			//Type Arrays
			//ARRAY OF BOOL
			IF FIND(Lynus_Standards.GVL_Communicator.arrInterfaceInfoAlVariables[byReadWriteArrayNumber,udiActiveNumberOfSymbol_ReadAds].sSymbolType,'OF BOOL') <> 0 THEN
				stADSRead_ReadAds[udiActiveNumberOfSymbol_ReadAds].sFullSymbolName := Lynus_Standards.GVL_Communicator.arrInterfaceInfoAlVariables[byReadWriteArrayNumber,udiActiveNumberOfSymbol_ReadAds].sFullSymbolName;
					stADSRead_ReadAds[udiActiveNumberOfSymbol_ReadAds].arrValue := arrValueDefault_ReadAds;	
						IF Lynus_Standards.GVL_Communicator.arrInterfaceInfoAlVariables[byReadWriteArrayNumber,udiActiveNumberOfSymbol_ReadAds].uiSizeArray <= Lynus_Standards.Constants_Communicator.bySizeOfValueArray THEN  
							FOR uiLPWriteValueByArray_ReadAds := 1 TO Lynus_Standards.GVL_Communicator.arrInterfaceInfoAlVariables[byReadWriteArrayNumber,udiActiveNumberOfSymbol_ReadAds].uiSizeArray BY 1 DO 	
								stADSRead_ReadAds[udiActiveNumberOfSymbol_ReadAds].arrValue[uiLPWriteValueByArray_ReadAds] := BYTE_TO_STRING(arrValueAfterRead_ReadAds[uiLPWriteValueByArray_ReadAds]);
							END_FOR 
						END_IF
			END_IF 
				//ARRAY OF BYTE
				IF FIND(Lynus_Standards.GVL_Communicator.arrInterfaceInfoAlVariables[byReadWriteArrayNumber,udiActiveNumberOfSymbol_ReadAds].sSymbolType,'OF BYTE') <> 0 THEN
					stADSRead_ReadAds[udiActiveNumberOfSymbol_ReadAds].sFullSymbolName := Lynus_Standards.GVL_Communicator.arrInterfaceInfoAlVariables[byReadWriteArrayNumber,udiActiveNumberOfSymbol_ReadAds].sFullSymbolName;
						stADSRead_ReadAds[udiActiveNumberOfSymbol_ReadAds].arrValue := arrValueDefault_ReadAds;	
							IF Lynus_Standards.GVL_Communicator.arrInterfaceInfoAlVariables[byReadWriteArrayNumber,udiActiveNumberOfSymbol_ReadAds].uiSizeArray <= Lynus_Standards.Constants_Communicator.bySizeOfValueArray THEN  
								FOR uiLPWriteValueByArray_ReadAds := 1 TO Lynus_Standards.GVL_Communicator.arrInterfaceInfoAlVariables[byReadWriteArrayNumber,udiActiveNumberOfSymbol_ReadAds].uiSizeArray BY 1 DO 	
									stADSRead_ReadAds[udiActiveNumberOfSymbol_ReadAds].arrValue[uiLPWriteValueByArray_ReadAds] := BYTE_TO_STRING(arrValueAfterRead_ReadAds[uiLPWriteValueByArray_ReadAds]);
								END_FOR 
							END_IF
				END_IF
			//ARRAY OF WORD
			IF FIND(Lynus_Standards.GVL_Communicator.arrInterfaceInfoAlVariables[byReadWriteArrayNumber,udiActiveNumberOfSymbol_ReadAds].sSymbolType,'OF WORD') <> 0 THEN
				stADSRead_ReadAds[udiActiveNumberOfSymbol_ReadAds].sFullSymbolName := Lynus_Standards.GVL_Communicator.arrInterfaceInfoAlVariables[byReadWriteArrayNumber,udiActiveNumberOfSymbol_ReadAds].sFullSymbolName;
					stADSRead_ReadAds[udiActiveNumberOfSymbol_ReadAds].arrValue := arrValueDefault_ReadAds;	
						IF Lynus_Standards.GVL_Communicator.arrInterfaceInfoAlVariables[byReadWriteArrayNumber,udiActiveNumberOfSymbol_ReadAds].uiSizeArray <= Lynus_Standards.Constants_Communicator.bySizeOfValueArray THEN  
							FOR uiLPWriteValueByArray_ReadAds := 1 TO Lynus_Standards.GVL_Communicator.arrInterfaceInfoAlVariables[byReadWriteArrayNumber,udiActiveNumberOfSymbol_ReadAds].uiSizeArray BY 1 DO
								arrCounterWriteValueInArray_ReadAds[1] := LIMIT(1,arrCounterWriteValueInArray_ReadAds[1],1600); arrCounterWriteValueInArray_ReadAds[2] := LIMIT(2,arrCounterWriteValueInArray_ReadAds[2],1600);
									stADSRead_ReadAds[udiActiveNumberOfSymbol_ReadAds].arrValue[uiLPWriteValueByArray_ReadAds] := WORD_TO_STRING(SHL(BYTE_TO_WORD(arrValueAfterRead_ReadAds[arrCounterWriteValueInArray_ReadAds[2]]),8) + BYTE_TO_WORD(arrValueAfterRead_ReadAds[arrCounterWriteValueInArray_ReadAds[1]]));;
								arrCounterWriteValueInArray_ReadAds[1] := arrCounterWriteValueInArray_ReadAds[1] + 2; arrCounterWriteValueInArray_ReadAds[2] := arrCounterWriteValueInArray_ReadAds[2] + 2;
							END_FOR 
						END_IF
			END_IF
				//ARRAY OF DWORD	
				IF FIND(Lynus_Standards.GVL_Communicator.arrInterfaceInfoAlVariables[byReadWriteArrayNumber,udiActiveNumberOfSymbol_ReadAds].sSymbolType,'OF DWORD') <> 0 THEN
					stADSRead_ReadAds[udiActiveNumberOfSymbol_ReadAds].sFullSymbolName := Lynus_Standards.GVL_Communicator.arrInterfaceInfoAlVariables[byReadWriteArrayNumber,udiActiveNumberOfSymbol_ReadAds].sFullSymbolName;
						stADSRead_ReadAds[udiActiveNumberOfSymbol_ReadAds].arrValue := arrValueDefault_ReadAds;	
							IF Lynus_Standards.GVL_Communicator.arrInterfaceInfoAlVariables[byReadWriteArrayNumber,udiActiveNumberOfSymbol_ReadAds].uiSizeArray <= Lynus_Standards.Constants_Communicator.bySizeOfValueArray THEN  
								FOR uiLPWriteValueByArray_ReadAds := 1 TO Lynus_Standards.GVL_Communicator.arrInterfaceInfoAlVariables[byReadWriteArrayNumber,udiActiveNumberOfSymbol_ReadAds].uiSizeArray BY 1 DO
									arrCounterWriteValueInArray_ReadAds[1] := LIMIT(1,arrCounterWriteValueInArray_ReadAds[1],1600); arrCounterWriteValueInArray_ReadAds[2] := LIMIT(2,arrCounterWriteValueInArray_ReadAds[2],1600);
										arrCounterWriteValueInArray_ReadAds[3] := LIMIT(3,arrCounterWriteValueInArray_ReadAds[3],1600); arrCounterWriteValueInArray_ReadAds[4] := LIMIT(4,arrCounterWriteValueInArray_ReadAds[4],1600);
											stADSRead_ReadAds[udiActiveNumberOfSymbol_ReadAds].arrValue[uiLPWriteValueByArray_ReadAds] := DWORD_TO_STRING(SHL(BYTE_TO_DWORD(arrValueAfterRead_ReadAds[arrCounterWriteValueInArray_ReadAds[4]]),24) + SHL(BYTE_TO_DWORD(arrValueAfterRead_ReadAds[arrCounterWriteValueInArray_ReadAds[3]]),16) + SHL(BYTE_TO_DWORD(arrValueAfterRead_ReadAds[arrCounterWriteValueInArray_ReadAds[2]]),8) + BYTE_TO_DWORD(arrValueAfterRead_ReadAds[arrCounterWriteValueInArray_ReadAds[1]]));
									arrCounterWriteValueInArray_ReadAds[1] := arrCounterWriteValueInArray_ReadAds[1] + 4; arrCounterWriteValueInArray_ReadAds[2] := arrCounterWriteValueInArray_ReadAds[2] + 4;
										arrCounterWriteValueInArray_ReadAds[3] := arrCounterWriteValueInArray_ReadAds[3] + 4; arrCounterWriteValueInArray_ReadAds[4] := arrCounterWriteValueInArray_ReadAds[4] + 4;
								END_FOR 
							END_IF
				END_IF
			//ARRAY OF SINT
			IF FIND(Lynus_Standards.GVL_Communicator.arrInterfaceInfoAlVariables[byReadWriteArrayNumber,udiActiveNumberOfSymbol_ReadAds].sSymbolType,'OF SINT') <> 0 THEN
				stADSRead_ReadAds[udiActiveNumberOfSymbol_ReadAds].sFullSymbolName := Lynus_Standards.GVL_Communicator.arrInterfaceInfoAlVariables[byReadWriteArrayNumber,udiActiveNumberOfSymbol_ReadAds].sFullSymbolName;
					stADSRead_ReadAds[udiActiveNumberOfSymbol_ReadAds].arrValue := arrValueDefault_ReadAds;	
						IF Lynus_Standards.GVL_Communicator.arrInterfaceInfoAlVariables[byReadWriteArrayNumber,udiActiveNumberOfSymbol_ReadAds].uiSizeArray <= Lynus_Standards.Constants_Communicator.bySizeOfValueArray THEN  
							FOR uiLPWriteValueByArray_ReadAds := 1 TO Lynus_Standards.GVL_Communicator.arrInterfaceInfoAlVariables[byReadWriteArrayNumber,udiActiveNumberOfSymbol_ReadAds].uiSizeArray BY 1 DO 	
								stADSRead_ReadAds[udiActiveNumberOfSymbol_ReadAds].arrValue[uiLPWriteValueByArray_ReadAds] := SINT_TO_STRING(BYTE_TO_SINT(arrValueAfterRead_ReadAds[uiLPWriteValueByArray_ReadAds]));
							END_FOR 
						END_IF
			END_IF
				//ARRAY OF USINT
				IF FIND(Lynus_Standards.GVL_Communicator.arrInterfaceInfoAlVariables[byReadWriteArrayNumber,udiActiveNumberOfSymbol_ReadAds].sSymbolType,'OF USINT') <> 0 THEN
					stADSRead_ReadAds[udiActiveNumberOfSymbol_ReadAds].sFullSymbolName := Lynus_Standards.GVL_Communicator.arrInterfaceInfoAlVariables[byReadWriteArrayNumber,udiActiveNumberOfSymbol_ReadAds].sFullSymbolName;
						stADSRead_ReadAds[udiActiveNumberOfSymbol_ReadAds].arrValue := arrValueDefault_ReadAds;	
							IF Lynus_Standards.GVL_Communicator.arrInterfaceInfoAlVariables[byReadWriteArrayNumber,udiActiveNumberOfSymbol_ReadAds].uiSizeArray <= Lynus_Standards.Constants_Communicator.bySizeOfValueArray THEN  
								FOR uiLPWriteValueByArray_ReadAds := 1 TO Lynus_Standards.GVL_Communicator.arrInterfaceInfoAlVariables[byReadWriteArrayNumber,udiActiveNumberOfSymbol_ReadAds].uiSizeArray BY 1 DO 	
									stADSRead_ReadAds[udiActiveNumberOfSymbol_ReadAds].arrValue[uiLPWriteValueByArray_ReadAds] := USINT_TO_STRING(BYTE_TO_USINT(arrValueAfterRead_ReadAds[uiLPWriteValueByArray_ReadAds]));
								END_FOR 
							END_IF
				END_IF
			//ARRAY OF INT
			IF FIND(Lynus_Standards.GVL_Communicator.arrInterfaceInfoAlVariables[byReadWriteArrayNumber,udiActiveNumberOfSymbol_ReadAds].sSymbolType,'OF INT') <> 0 THEN
				stADSRead_ReadAds[udiActiveNumberOfSymbol_ReadAds].sFullSymbolName := Lynus_Standards.GVL_Communicator.arrInterfaceInfoAlVariables[byReadWriteArrayNumber,udiActiveNumberOfSymbol_ReadAds].sFullSymbolName;
					stADSRead_ReadAds[udiActiveNumberOfSymbol_ReadAds].arrValue := arrValueDefault_ReadAds;	
						IF Lynus_Standards.GVL_Communicator.arrInterfaceInfoAlVariables[byReadWriteArrayNumber,udiActiveNumberOfSymbol_ReadAds].uiSizeArray <= Lynus_Standards.Constants_Communicator.bySizeOfValueArray THEN  
							FOR uiLPWriteValueByArray_ReadAds := 1 TO Lynus_Standards.GVL_Communicator.arrInterfaceInfoAlVariables[byReadWriteArrayNumber,udiActiveNumberOfSymbol_ReadAds].uiSizeArray BY 1 DO
								arrCounterWriteValueInArray_ReadAds[1] := LIMIT(1,arrCounterWriteValueInArray_ReadAds[1],1600); arrCounterWriteValueInArray_ReadAds[2] := LIMIT(2,arrCounterWriteValueInArray_ReadAds[2],1600);
									stADSRead_ReadAds[udiActiveNumberOfSymbol_ReadAds].arrValue[uiLPWriteValueByArray_ReadAds] := INT_TO_STRING(SHL(BYTE_TO_INT(arrValueAfterRead_ReadAds[arrCounterWriteValueInArray_ReadAds[2]]),8) + BYTE_TO_INT(arrValueAfterRead_ReadAds[arrCounterWriteValueInArray_ReadAds[1]]));;
								arrCounterWriteValueInArray_ReadAds[1] := arrCounterWriteValueInArray_ReadAds[1] + 2; arrCounterWriteValueInArray_ReadAds[2] := arrCounterWriteValueInArray_ReadAds[2] + 2;
							END_FOR 
						END_IF
			END_IF
				//ARRAY OF UINT
				IF FIND(Lynus_Standards.GVL_Communicator.arrInterfaceInfoAlVariables[byReadWriteArrayNumber,udiActiveNumberOfSymbol_ReadAds].sSymbolType,'OF UINT') <> 0 THEN
					stADSRead_ReadAds[udiActiveNumberOfSymbol_ReadAds].sFullSymbolName := Lynus_Standards.GVL_Communicator.arrInterfaceInfoAlVariables[byReadWriteArrayNumber,udiActiveNumberOfSymbol_ReadAds].sFullSymbolName;
						stADSRead_ReadAds[udiActiveNumberOfSymbol_ReadAds].arrValue := arrValueDefault_ReadAds;	
							IF Lynus_Standards.GVL_Communicator.arrInterfaceInfoAlVariables[byReadWriteArrayNumber,udiActiveNumberOfSymbol_ReadAds].uiSizeArray <= Lynus_Standards.Constants_Communicator.bySizeOfValueArray THEN  
								FOR uiLPWriteValueByArray_ReadAds := 1 TO Lynus_Standards.GVL_Communicator.arrInterfaceInfoAlVariables[byReadWriteArrayNumber,udiActiveNumberOfSymbol_ReadAds].uiSizeArray BY 1 DO
									arrCounterWriteValueInArray_ReadAds[1] := LIMIT(1,arrCounterWriteValueInArray_ReadAds[1],1600); arrCounterWriteValueInArray_ReadAds[2] := LIMIT(2,arrCounterWriteValueInArray_ReadAds[2],1600);
										stADSRead_ReadAds[udiActiveNumberOfSymbol_ReadAds].arrValue[uiLPWriteValueByArray_ReadAds] := UINT_TO_STRING(SHL(BYTE_TO_UINT(arrValueAfterRead_ReadAds[arrCounterWriteValueInArray_ReadAds[2]]),8) + BYTE_TO_UINT(arrValueAfterRead_ReadAds[arrCounterWriteValueInArray_ReadAds[1]]));;
									arrCounterWriteValueInArray_ReadAds[1] := arrCounterWriteValueInArray_ReadAds[1] + 2; arrCounterWriteValueInArray_ReadAds[2] := arrCounterWriteValueInArray_ReadAds[2] + 2;
								END_FOR 
							END_IF
				END_IF
			//ARRAY OF DINT	
			IF FIND(Lynus_Standards.GVL_Communicator.arrInterfaceInfoAlVariables[byReadWriteArrayNumber,udiActiveNumberOfSymbol_ReadAds].sSymbolType,'OF DINT') <> 0 THEN
				stADSRead_ReadAds[udiActiveNumberOfSymbol_ReadAds].sFullSymbolName := Lynus_Standards.GVL_Communicator.arrInterfaceInfoAlVariables[byReadWriteArrayNumber,udiActiveNumberOfSymbol_ReadAds].sFullSymbolName;
					stADSRead_ReadAds[udiActiveNumberOfSymbol_ReadAds].arrValue := arrValueDefault_ReadAds;	
						IF Lynus_Standards.GVL_Communicator.arrInterfaceInfoAlVariables[byReadWriteArrayNumber,udiActiveNumberOfSymbol_ReadAds].uiSizeArray <= Lynus_Standards.Constants_Communicator.bySizeOfValueArray THEN  
							FOR uiLPWriteValueByArray_ReadAds := 1 TO Lynus_Standards.GVL_Communicator.arrInterfaceInfoAlVariables[byReadWriteArrayNumber,udiActiveNumberOfSymbol_ReadAds].uiSizeArray BY 1 DO
								arrCounterWriteValueInArray_ReadAds[1] := LIMIT(1,arrCounterWriteValueInArray_ReadAds[1],1600); arrCounterWriteValueInArray_ReadAds[2] := LIMIT(2,arrCounterWriteValueInArray_ReadAds[2],1600);
									arrCounterWriteValueInArray_ReadAds[3] := LIMIT(3,arrCounterWriteValueInArray_ReadAds[3],1600); arrCounterWriteValueInArray_ReadAds[4] := LIMIT(4,arrCounterWriteValueInArray_ReadAds[4],1600);
										stADSRead_ReadAds[udiActiveNumberOfSymbol_ReadAds].arrValue[uiLPWriteValueByArray_ReadAds] := DINT_TO_STRING(SHL(BYTE_TO_DINT(arrValueAfterRead_ReadAds[arrCounterWriteValueInArray_ReadAds[4]]),24) + SHL(BYTE_TO_DINT(arrValueAfterRead_ReadAds[arrCounterWriteValueInArray_ReadAds[3]]),16) + SHL(BYTE_TO_DINT(arrValueAfterRead_ReadAds[arrCounterWriteValueInArray_ReadAds[2]]),8) + BYTE_TO_DINT(arrValueAfterRead_ReadAds[arrCounterWriteValueInArray_ReadAds[1]]));
								arrCounterWriteValueInArray_ReadAds[1] := arrCounterWriteValueInArray_ReadAds[1] + 4; arrCounterWriteValueInArray_ReadAds[2] := arrCounterWriteValueInArray_ReadAds[2] + 4;
									arrCounterWriteValueInArray_ReadAds[3] := arrCounterWriteValueInArray_ReadAds[3] + 4; arrCounterWriteValueInArray_ReadAds[4] := arrCounterWriteValueInArray_ReadAds[4] + 4;
							END_FOR 
						END_IF
			END_IF
				//ARRAY OF UDINT	
				IF FIND(Lynus_Standards.GVL_Communicator.arrInterfaceInfoAlVariables[byReadWriteArrayNumber,udiActiveNumberOfSymbol_ReadAds].sSymbolType,'OF UDINT') <> 0 THEN
					stADSRead_ReadAds[udiActiveNumberOfSymbol_ReadAds].sFullSymbolName := Lynus_Standards.GVL_Communicator.arrInterfaceInfoAlVariables[byReadWriteArrayNumber,udiActiveNumberOfSymbol_ReadAds].sFullSymbolName;
						stADSRead_ReadAds[udiActiveNumberOfSymbol_ReadAds].arrValue := arrValueDefault_ReadAds;	
							IF Lynus_Standards.GVL_Communicator.arrInterfaceInfoAlVariables[byReadWriteArrayNumber,udiActiveNumberOfSymbol_ReadAds].uiSizeArray <= Lynus_Standards.Constants_Communicator.bySizeOfValueArray THEN  
								FOR uiLPWriteValueByArray_ReadAds := 1 TO Lynus_Standards.GVL_Communicator.arrInterfaceInfoAlVariables[byReadWriteArrayNumber,udiActiveNumberOfSymbol_ReadAds].uiSizeArray BY 1 DO
									arrCounterWriteValueInArray_ReadAds[1] := LIMIT(1,arrCounterWriteValueInArray_ReadAds[1],1600); arrCounterWriteValueInArray_ReadAds[2] := LIMIT(2,arrCounterWriteValueInArray_ReadAds[2],1600);
										arrCounterWriteValueInArray_ReadAds[3] := LIMIT(3,arrCounterWriteValueInArray_ReadAds[3],1600); arrCounterWriteValueInArray_ReadAds[4] := LIMIT(4,arrCounterWriteValueInArray_ReadAds[4],1600);
											stADSRead_ReadAds[udiActiveNumberOfSymbol_ReadAds].arrValue[uiLPWriteValueByArray_ReadAds] := UDINT_TO_STRING(SHL(BYTE_TO_UDINT(arrValueAfterRead_ReadAds[arrCounterWriteValueInArray_ReadAds[4]]),24) + SHL(BYTE_TO_UDINT(arrValueAfterRead_ReadAds[arrCounterWriteValueInArray_ReadAds[3]]),16) + SHL(BYTE_TO_UDINT(arrValueAfterRead_ReadAds[arrCounterWriteValueInArray_ReadAds[2]]),8) + BYTE_TO_UDINT(arrValueAfterRead_ReadAds[arrCounterWriteValueInArray_ReadAds[1]]));
									arrCounterWriteValueInArray_ReadAds[1] := arrCounterWriteValueInArray_ReadAds[1] + 4; arrCounterWriteValueInArray_ReadAds[2] := arrCounterWriteValueInArray_ReadAds[2] + 4;
										arrCounterWriteValueInArray_ReadAds[3] := arrCounterWriteValueInArray_ReadAds[3] + 4; arrCounterWriteValueInArray_ReadAds[4] := arrCounterWriteValueInArray_ReadAds[4] + 4;
								END_FOR 
							END_IF
				END_IF
					//ARRAY OF LINT	
					IF FIND(Lynus_Standards.GVL_Communicator.arrInterfaceInfoAlVariables[byReadWriteArrayNumber,udiActiveNumberOfSymbol_ReadAds].sSymbolType,'OF LINT') <> 0 THEN
						stADSRead_ReadAds[udiActiveNumberOfSymbol_ReadAds].sFullSymbolName := Lynus_Standards.GVL_Communicator.arrInterfaceInfoAlVariables[byReadWriteArrayNumber,udiActiveNumberOfSymbol_ReadAds].sFullSymbolName;
							stADSRead_ReadAds[udiActiveNumberOfSymbol_ReadAds].arrValue := arrValueDefault_ReadAds;	
								IF Lynus_Standards.GVL_Communicator.arrInterfaceInfoAlVariables[byReadWriteArrayNumber,udiActiveNumberOfSymbol_ReadAds].uiSizeArray <= Lynus_Standards.Constants_Communicator.bySizeOfValueArray THEN  
									FOR uiLPWriteValueByArray_ReadAds := 1 TO Lynus_Standards.GVL_Communicator.arrInterfaceInfoAlVariables[byReadWriteArrayNumber,udiActiveNumberOfSymbol_ReadAds].uiSizeArray BY 1 DO
										arrCounterWriteValueInArray_ReadAds[1] := LIMIT(1,arrCounterWriteValueInArray_ReadAds[1],1600); arrCounterWriteValueInArray_ReadAds[2] := LIMIT(2,arrCounterWriteValueInArray_ReadAds[2],1600);
											arrCounterWriteValueInArray_ReadAds[3] := LIMIT(3,arrCounterWriteValueInArray_ReadAds[3],1600); arrCounterWriteValueInArray_ReadAds[4] := LIMIT(4,arrCounterWriteValueInArray_ReadAds[4],1600);
												arrCounterWriteValueInArray_ReadAds[5] := LIMIT(5,arrCounterWriteValueInArray_ReadAds[5],1600); arrCounterWriteValueInArray_ReadAds[6] := LIMIT(6,arrCounterWriteValueInArray_ReadAds[6],1600);
													arrCounterWriteValueInArray_ReadAds[7] := LIMIT(7,arrCounterWriteValueInArray_ReadAds[7],1600); arrCounterWriteValueInArray_ReadAds[8] := LIMIT(8,arrCounterWriteValueInArray_ReadAds[8],1600);
														stADSRead_ReadAds[udiActiveNumberOfSymbol_ReadAds].arrValue[uiLPWriteValueByArray_ReadAds] := LINT_TO_STRING(SHL(BYTE_TO_LINT(arrValueAfterRead_ReadAds[arrCounterWriteValueInArray_ReadAds[8]]),56) + SHL(BYTE_TO_LINT(arrValueAfterRead_ReadAds[arrCounterWriteValueInArray_ReadAds[7]]),48) + SHL(BYTE_TO_LINT(arrValueAfterRead_ReadAds[arrCounterWriteValueInArray_ReadAds[6]]),40) + SHL(BYTE_TO_LINT(arrValueAfterRead_ReadAds[arrCounterWriteValueInArray_ReadAds[5]]),32) +
																																							SHL(BYTE_TO_LINT(arrValueAfterRead_ReadAds[arrCounterWriteValueInArray_ReadAds[4]]),24) + SHL(BYTE_TO_LINT(arrValueAfterRead_ReadAds[arrCounterWriteValueInArray_ReadAds[3]]),16) + SHL(BYTE_TO_LINT(arrValueAfterRead_ReadAds[arrCounterWriteValueInArray_ReadAds[2]]),8) + BYTE_TO_LINT(arrValueAfterRead_ReadAds[arrCounterWriteValueInArray_ReadAds[1]]));
										arrCounterWriteValueInArray_ReadAds[1] := arrCounterWriteValueInArray_ReadAds[1] + 8; arrCounterWriteValueInArray_ReadAds[2] := arrCounterWriteValueInArray_ReadAds[2] + 8;
											arrCounterWriteValueInArray_ReadAds[3] := arrCounterWriteValueInArray_ReadAds[3] + 8; arrCounterWriteValueInArray_ReadAds[4] := arrCounterWriteValueInArray_ReadAds[4] + 8;
												arrCounterWriteValueInArray_ReadAds[5] := arrCounterWriteValueInArray_ReadAds[5] + 8; arrCounterWriteValueInArray_ReadAds[6] := arrCounterWriteValueInArray_ReadAds[6] + 8;
													arrCounterWriteValueInArray_ReadAds[7] := arrCounterWriteValueInArray_ReadAds[7] + 8; arrCounterWriteValueInArray_ReadAds[8] := arrCounterWriteValueInArray_ReadAds[8] + 8;
									END_FOR 
								END_IF
					END_IF
				//ARRAY OF ULINT	
				IF FIND(Lynus_Standards.GVL_Communicator.arrInterfaceInfoAlVariables[byReadWriteArrayNumber,udiActiveNumberOfSymbol_ReadAds].sSymbolType,'OF ULINT') <> 0 THEN
					stADSRead_ReadAds[udiActiveNumberOfSymbol_ReadAds].sFullSymbolName := Lynus_Standards.GVL_Communicator.arrInterfaceInfoAlVariables[byReadWriteArrayNumber,udiActiveNumberOfSymbol_ReadAds].sFullSymbolName;
						stADSRead_ReadAds[udiActiveNumberOfSymbol_ReadAds].arrValue := arrValueDefault_ReadAds;	
							IF Lynus_Standards.GVL_Communicator.arrInterfaceInfoAlVariables[byReadWriteArrayNumber,udiActiveNumberOfSymbol_ReadAds].uiSizeArray <= Lynus_Standards.Constants_Communicator.bySizeOfValueArray THEN  
								FOR uiLPWriteValueByArray_ReadAds := 1 TO Lynus_Standards.GVL_Communicator.arrInterfaceInfoAlVariables[byReadWriteArrayNumber,udiActiveNumberOfSymbol_ReadAds].uiSizeArray BY 1 DO
									arrCounterWriteValueInArray_ReadAds[1] := LIMIT(1,arrCounterWriteValueInArray_ReadAds[1],1600); arrCounterWriteValueInArray_ReadAds[2] := LIMIT(2,arrCounterWriteValueInArray_ReadAds[2],1600);
										arrCounterWriteValueInArray_ReadAds[3] := LIMIT(3,arrCounterWriteValueInArray_ReadAds[3],1600); arrCounterWriteValueInArray_ReadAds[4] := LIMIT(4,arrCounterWriteValueInArray_ReadAds[4],1600);
											arrCounterWriteValueInArray_ReadAds[5] := LIMIT(5,arrCounterWriteValueInArray_ReadAds[5],1600); arrCounterWriteValueInArray_ReadAds[6] := LIMIT(6,arrCounterWriteValueInArray_ReadAds[6],1600);
												arrCounterWriteValueInArray_ReadAds[7] := LIMIT(7,arrCounterWriteValueInArray_ReadAds[7],1600); arrCounterWriteValueInArray_ReadAds[8] := LIMIT(8,arrCounterWriteValueInArray_ReadAds[8],1600);
													stADSRead_ReadAds[udiActiveNumberOfSymbol_ReadAds].arrValue[uiLPWriteValueByArray_ReadAds] := ULINT_TO_STRING(SHL(BYTE_TO_ULINT(arrValueAfterRead_ReadAds[arrCounterWriteValueInArray_ReadAds[8]]),56) + SHL(BYTE_TO_ULINT(arrValueAfterRead_ReadAds[arrCounterWriteValueInArray_ReadAds[7]]),48) + SHL(BYTE_TO_ULINT(arrValueAfterRead_ReadAds[arrCounterWriteValueInArray_ReadAds[6]]),40) + SHL(BYTE_TO_ULINT(arrValueAfterRead_ReadAds[arrCounterWriteValueInArray_ReadAds[5]]),32) +
																																						SHL(BYTE_TO_ULINT(arrValueAfterRead_ReadAds[arrCounterWriteValueInArray_ReadAds[4]]),24) + SHL(BYTE_TO_ULINT(arrValueAfterRead_ReadAds[arrCounterWriteValueInArray_ReadAds[3]]),16) + SHL(BYTE_TO_ULINT(arrValueAfterRead_ReadAds[arrCounterWriteValueInArray_ReadAds[2]]),8) + BYTE_TO_ULINT(arrValueAfterRead_ReadAds[arrCounterWriteValueInArray_ReadAds[1]]));
									arrCounterWriteValueInArray_ReadAds[1] := arrCounterWriteValueInArray_ReadAds[1] + 8; arrCounterWriteValueInArray_ReadAds[2] := arrCounterWriteValueInArray_ReadAds[2] + 8;
										arrCounterWriteValueInArray_ReadAds[3] := arrCounterWriteValueInArray_ReadAds[3] + 8; arrCounterWriteValueInArray_ReadAds[4] := arrCounterWriteValueInArray_ReadAds[4] + 8;
											arrCounterWriteValueInArray_ReadAds[5] := arrCounterWriteValueInArray_ReadAds[5] + 8; arrCounterWriteValueInArray_ReadAds[6] := arrCounterWriteValueInArray_ReadAds[6] + 8;
												arrCounterWriteValueInArray_ReadAds[7] := arrCounterWriteValueInArray_ReadAds[7] + 8; arrCounterWriteValueInArray_ReadAds[8] := arrCounterWriteValueInArray_ReadAds[8] + 8;
								END_FOR 
							END_IF
				END_IF
					//ARRAY OF LWORD	
					IF FIND(Lynus_Standards.GVL_Communicator.arrInterfaceInfoAlVariables[byReadWriteArrayNumber,udiActiveNumberOfSymbol_ReadAds].sSymbolType,'OF LWORD') <> 0 THEN
						stADSRead_ReadAds[udiActiveNumberOfSymbol_ReadAds].sFullSymbolName := Lynus_Standards.GVL_Communicator.arrInterfaceInfoAlVariables[byReadWriteArrayNumber,udiActiveNumberOfSymbol_ReadAds].sFullSymbolName;
							stADSRead_ReadAds[udiActiveNumberOfSymbol_ReadAds].arrValue := arrValueDefault_ReadAds;	
								IF Lynus_Standards.GVL_Communicator.arrInterfaceInfoAlVariables[byReadWriteArrayNumber,udiActiveNumberOfSymbol_ReadAds].uiSizeArray <= Lynus_Standards.Constants_Communicator.bySizeOfValueArray THEN  
									FOR uiLPWriteValueByArray_ReadAds := 1 TO Lynus_Standards.GVL_Communicator.arrInterfaceInfoAlVariables[byReadWriteArrayNumber,udiActiveNumberOfSymbol_ReadAds].uiSizeArray BY 1 DO
										arrCounterWriteValueInArray_ReadAds[1] := LIMIT(1,arrCounterWriteValueInArray_ReadAds[1],1600); arrCounterWriteValueInArray_ReadAds[2] := LIMIT(2,arrCounterWriteValueInArray_ReadAds[2],1600);
											arrCounterWriteValueInArray_ReadAds[3] := LIMIT(3,arrCounterWriteValueInArray_ReadAds[3],1600); arrCounterWriteValueInArray_ReadAds[4] := LIMIT(4,arrCounterWriteValueInArray_ReadAds[4],1600);
												arrCounterWriteValueInArray_ReadAds[5] := LIMIT(5,arrCounterWriteValueInArray_ReadAds[5],1600); arrCounterWriteValueInArray_ReadAds[6] := LIMIT(6,arrCounterWriteValueInArray_ReadAds[6],1600);
													arrCounterWriteValueInArray_ReadAds[7] := LIMIT(7,arrCounterWriteValueInArray_ReadAds[7],1600); arrCounterWriteValueInArray_ReadAds[8] := LIMIT(8,arrCounterWriteValueInArray_ReadAds[8],1600);
														stADSRead_ReadAds[udiActiveNumberOfSymbol_ReadAds].arrValue[uiLPWriteValueByArray_ReadAds] := LWORD_TO_STRING(SHL(BYTE_TO_LWORD(arrValueAfterRead_ReadAds[arrCounterWriteValueInArray_ReadAds[8]]),56) + SHL(BYTE_TO_LWORD(arrValueAfterRead_ReadAds[arrCounterWriteValueInArray_ReadAds[7]]),48) + SHL(BYTE_TO_LWORD(arrValueAfterRead_ReadAds[arrCounterWriteValueInArray_ReadAds[6]]),40) + SHL(BYTE_TO_LWORD(arrValueAfterRead_ReadAds[arrCounterWriteValueInArray_ReadAds[5]]),32) +
																																							SHL(BYTE_TO_LWORD(arrValueAfterRead_ReadAds[arrCounterWriteValueInArray_ReadAds[4]]),24) + SHL(BYTE_TO_LWORD(arrValueAfterRead_ReadAds[arrCounterWriteValueInArray_ReadAds[3]]),16) + SHL(BYTE_TO_LWORD(arrValueAfterRead_ReadAds[arrCounterWriteValueInArray_ReadAds[2]]),8) + BYTE_TO_LWORD(arrValueAfterRead_ReadAds[arrCounterWriteValueInArray_ReadAds[1]]));
										arrCounterWriteValueInArray_ReadAds[1] := arrCounterWriteValueInArray_ReadAds[1] + 8; arrCounterWriteValueInArray_ReadAds[2] := arrCounterWriteValueInArray_ReadAds[2] + 8;
											arrCounterWriteValueInArray_ReadAds[3] := arrCounterWriteValueInArray_ReadAds[3] + 8; arrCounterWriteValueInArray_ReadAds[4] := arrCounterWriteValueInArray_ReadAds[4] + 8;
												arrCounterWriteValueInArray_ReadAds[5] := arrCounterWriteValueInArray_ReadAds[5] + 8; arrCounterWriteValueInArray_ReadAds[6] := arrCounterWriteValueInArray_ReadAds[6] + 8;
													arrCounterWriteValueInArray_ReadAds[7] := arrCounterWriteValueInArray_ReadAds[7] + 8; arrCounterWriteValueInArray_ReadAds[8] := arrCounterWriteValueInArray_ReadAds[8] + 8;
									END_FOR 
								END_IF
					END_IF
				//ARRAY OF REAL
				IF FIND(Lynus_Standards.GVL_Communicator.arrInterfaceInfoAlVariables[byReadWriteArrayNumber,udiActiveNumberOfSymbol_ReadAds].sSymbolType,'OF REAL') <> 0 THEN
					stADSRead_ReadAds[udiActiveNumberOfSymbol_ReadAds].sFullSymbolName := Lynus_Standards.GVL_Communicator.arrInterfaceInfoAlVariables[byReadWriteArrayNumber,udiActiveNumberOfSymbol_ReadAds].sFullSymbolName;
						stADSRead_ReadAds[udiActiveNumberOfSymbol_ReadAds].arrValue := arrValueDefault_ReadAds;	
							IF Lynus_Standards.GVL_Communicator.arrInterfaceInfoAlVariables[byReadWriteArrayNumber,udiActiveNumberOfSymbol_ReadAds].uiSizeArray <= Lynus_Standards.Constants_Communicator.bySizeOfValueArray THEN  
								FOR uiLPWriteValueByArray_ReadAds := 1 TO Lynus_Standards.GVL_Communicator.arrInterfaceInfoAlVariables[byReadWriteArrayNumber,udiActiveNumberOfSymbol_ReadAds].uiSizeArray BY 1 DO
									arrCounterWriteValueInArray_ReadAds[1] := LIMIT(1,arrCounterWriteValueInArray_ReadAds[1],1600); arrCounterWriteValueInArray_ReadAds[2] := LIMIT(2,arrCounterWriteValueInArray_ReadAds[2],1600);
										arrCounterWriteValueInArray_ReadAds[3] := LIMIT(3,arrCounterWriteValueInArray_ReadAds[3],1600); arrCounterWriteValueInArray_ReadAds[4] := LIMIT(4,arrCounterWriteValueInArray_ReadAds[4],1600);
											unConvertDWORD_TO_REAL_ReadAds.dwRawValue := DINT_TO_DWORD(DWORD_TO_DINT(SHL(BYTE_TO_DWORD(arrValueAfterRead_ReadAds[arrCounterWriteValueInArray_ReadAds[4]]),24) + SHL(BYTE_TO_DWORD(arrValueAfterRead_ReadAds[arrCounterWriteValueInArray_ReadAds[3]]),16) + SHL(BYTE_TO_DWORD(arrValueAfterRead_ReadAds[arrCounterWriteValueInArray_ReadAds[2]]),8) + BYTE_TO_DWORD(arrValueAfterRead_ReadAds[arrCounterWriteValueInArray_ReadAds[1]])));
									arrCounterWriteValueInArray_ReadAds[1] := arrCounterWriteValueInArray_ReadAds[1] + 4; arrCounterWriteValueInArray_ReadAds[2] := arrCounterWriteValueInArray_ReadAds[2] + 4;
										arrCounterWriteValueInArray_ReadAds[3] := arrCounterWriteValueInArray_ReadAds[3] + 4; arrCounterWriteValueInArray_ReadAds[4] := arrCounterWriteValueInArray_ReadAds[4] + 4;					
											IF IsFinite(F_REAL(unConvertDWORD_TO_REAL_ReadAds.rValueFloat)) THEN 
												IF LEN(REAL_TO_STRING(unConvertDWORD_TO_REAL_ReadAds.rValueFloat)) <= 30 THEN 
													IF FIND(REAL_TO_STRING(unConvertDWORD_TO_REAL_ReadAds.rValueFloat),'e') = 0 AND FIND(REAL_TO_STRING(unConvertDWORD_TO_REAL_ReadAds.rValueFloat),'E') = 0 THEN 
														sStringFloat_ReadAds := REAL_TO_STRING(unConvertDWORD_TO_REAL_ReadAds.rValueFloat);
															iFindPointFloat_ReadAds := FIND(sStringFloat_ReadAds,'.');
																sStringFloat_ReadAds := DELETE(sStringFloat_ReadAds,iFindPointFloat_ReadAds,1);
																	iPrecision_ReadAds := LEN(sStringFloat_ReadAds);
																		iPrecision_ReadAds := LIMIT(0,iPrecision_ReadAds,8);
														IF LEN(LREAL_TO_FMTSTR(REAL_TO_LREAL(unConvertDWORD_TO_REAL_ReadAds.rValueFloat),iPrecision_ReadAds,TRUE)) <= 30 THEN	 			
															//Check if the output from Function LREAL_TO_FMTSTR is ok 
															IF LREAL_TO_FMTSTR(REAL_TO_LREAL(unConvertDWORD_TO_REAL_ReadAds.rValueFloat),iPrecision_ReadAds,TRUE) <> '#INF' AND LREAL_TO_FMTSTR(REAL_TO_LREAL(unConvertDWORD_TO_REAL_ReadAds.rValueFloat),iPrecision_ReadAds,TRUE) <> '-#INF' AND
																LREAL_TO_FMTSTR(REAL_TO_LREAL(unConvertDWORD_TO_REAL_ReadAds.rValueFloat),iPrecision_ReadAds,TRUE) <> '#QNAN' AND LREAL_TO_FMTSTR(REAL_TO_LREAL(unConvertDWORD_TO_REAL_ReadAds.rValueFloat),iPrecision_ReadAds,TRUE) <> '-#QNAN' AND
																	LREAL_TO_FMTSTR(REAL_TO_LREAL(unConvertDWORD_TO_REAL_ReadAds.rValueFloat),iPrecision_ReadAds,TRUE) <> '#OVF' AND LREAL_TO_FMTSTR(REAL_TO_LREAL(unConvertDWORD_TO_REAL_ReadAds.rValueFloat),iPrecision_ReadAds,TRUE) <> '-#OVF' THEN	   	 			
																		stADSRead_ReadAds[udiActiveNumberOfSymbol_ReadAds].arrValue[uiLPWriteValueByArray_ReadAds] := LREAL_TO_FMTSTR(REAL_TO_LREAL(unConvertDWORD_TO_REAL_ReadAds.rValueFloat),iPrecision_ReadAds,TRUE);
															ELSE
																iState_ReadAds := 200;
																	uiInternError_ReadAds := 1;
															END_IF
														ELSE
															//Check if the output from Function LREAL_TO_FMTSTR is ok 
															IF MID(LREAL_TO_FMTSTR(REAL_TO_LREAL(unConvertDWORD_TO_REAL_ReadAds.rValueFloat),iPrecision_ReadAds,TRUE),30,1) <> '#INF' AND MID(LREAL_TO_FMTSTR(REAL_TO_LREAL(unConvertDWORD_TO_REAL_ReadAds.rValueFloat),iPrecision_ReadAds,TRUE),30,1) <> '-#INF' AND
																MID(LREAL_TO_FMTSTR(REAL_TO_LREAL(unConvertDWORD_TO_REAL_ReadAds.rValueFloat),iPrecision_ReadAds,TRUE),30,1) <> '#QNAN' AND MID(LREAL_TO_FMTSTR(REAL_TO_LREAL(unConvertDWORD_TO_REAL_ReadAds.rValueFloat),iPrecision_ReadAds,TRUE),30,1) <> '-#QNAN' AND
																	MID(LREAL_TO_FMTSTR(REAL_TO_LREAL(unConvertDWORD_TO_REAL_ReadAds.rValueFloat),iPrecision_ReadAds,TRUE),30,1) <> '#OVF' AND MID(LREAL_TO_FMTSTR(REAL_TO_LREAL(unConvertDWORD_TO_REAL_ReadAds.rValueFloat),iPrecision_ReadAds,TRUE),30,1) <> '-#OVF' THEN 
																		stADSRead_ReadAds[udiActiveNumberOfSymbol_ReadAds].arrValue[uiLPWriteValueByArray_ReadAds] := MID(LREAL_TO_FMTSTR(REAL_TO_LREAL(unConvertDWORD_TO_REAL_ReadAds.rValueFloat),iPrecision_ReadAds,TRUE),30,1);
															ELSE
																iState_ReadAds := 200;
																	uiInternError_ReadAds := 1;
															END_IF
														END_IF
													ELSE
														stADSRead_ReadAds[udiActiveNumberOfSymbol_ReadAds].arrValue[uiLPWriteValueByArray_ReadAds] := REAL_TO_STRING(unConvertDWORD_TO_REAL_ReadAds.rValueFloat);
													END_IF 
												ELSE
													iState_ReadAds := 200;
														uiInternError_ReadAds := 1;
												END_IF
											ELSE
												iState_ReadAds := 200;
													uiInternError_ReadAds := 1;	
											END_IF
								END_FOR 
							END_IF
				END_IF
					//ARRAY OF LREAL
					IF FIND(Lynus_Standards.GVL_Communicator.arrInterfaceInfoAlVariables[byReadWriteArrayNumber,udiActiveNumberOfSymbol_ReadAds].sSymbolType,'OF LREAL') <> 0 THEN
						stADSRead_ReadAds[udiActiveNumberOfSymbol_ReadAds].sFullSymbolName := Lynus_Standards.GVL_Communicator.arrInterfaceInfoAlVariables[byReadWriteArrayNumber,udiActiveNumberOfSymbol_ReadAds].sFullSymbolName;
							stADSRead_ReadAds[udiActiveNumberOfSymbol_ReadAds].arrValue := arrValueDefault_ReadAds;	
								IF Lynus_Standards.GVL_Communicator.arrInterfaceInfoAlVariables[byReadWriteArrayNumber,udiActiveNumberOfSymbol_ReadAds].uiSizeArray <= Lynus_Standards.Constants_Communicator.bySizeOfValueArray THEN  
									FOR uiLPWriteValueByArray_ReadAds := 1 TO Lynus_Standards.GVL_Communicator.arrInterfaceInfoAlVariables[byReadWriteArrayNumber,udiActiveNumberOfSymbol_ReadAds].uiSizeArray BY 1 DO
										arrCounterWriteValueInArray_ReadAds[1] := LIMIT(1,arrCounterWriteValueInArray_ReadAds[1],1600); arrCounterWriteValueInArray_ReadAds[2] := LIMIT(2,arrCounterWriteValueInArray_ReadAds[2],1600);
											arrCounterWriteValueInArray_ReadAds[3] := LIMIT(3,arrCounterWriteValueInArray_ReadAds[3],1600); arrCounterWriteValueInArray_ReadAds[4] := LIMIT(4,arrCounterWriteValueInArray_ReadAds[4],1600);
												arrCounterWriteValueInArray_ReadAds[5] := LIMIT(5,arrCounterWriteValueInArray_ReadAds[5],1600); arrCounterWriteValueInArray_ReadAds[6] := LIMIT(6,arrCounterWriteValueInArray_ReadAds[6],1600);
													arrCounterWriteValueInArray_ReadAds[7] := LIMIT(7,arrCounterWriteValueInArray_ReadAds[7],1600); arrCounterWriteValueInArray_ReadAds[8] := LIMIT(8,arrCounterWriteValueInArray_ReadAds[8],1600);
														unConvertULINT_TO_LREAL_ReadAds.uliRawValue := LINT_TO_ULINT(ULINT_TO_LINT(SHL(BYTE_TO_ULINT(arrValueAfterRead_ReadAds[arrCounterWriteValueInArray_ReadAds[8]]),56) + SHL(BYTE_TO_ULINT(arrValueAfterRead_ReadAds[arrCounterWriteValueInArray_ReadAds[7]]),48) + SHL(BYTE_TO_ULINT(arrValueAfterRead_ReadAds[arrCounterWriteValueInArray_ReadAds[6]]),40) + SHL(BYTE_TO_ULINT(arrValueAfterRead_ReadAds[arrCounterWriteValueInArray_ReadAds[5]]),32) +
																											SHL(BYTE_TO_ULINT(arrValueAfterRead_ReadAds[arrCounterWriteValueInArray_ReadAds[4]]),24) + SHL(BYTE_TO_ULINT(arrValueAfterRead_ReadAds[arrCounterWriteValueInArray_ReadAds[3]]),16) + SHL(BYTE_TO_ULINT(arrValueAfterRead_ReadAds[arrCounterWriteValueInArray_ReadAds[2]]),8) + BYTE_TO_ULINT(arrValueAfterRead_ReadAds[arrCounterWriteValueInArray_ReadAds[1]])));
										arrCounterWriteValueInArray_ReadAds[1] := arrCounterWriteValueInArray_ReadAds[1] + 8; arrCounterWriteValueInArray_ReadAds[2] := arrCounterWriteValueInArray_ReadAds[2] + 8;
											arrCounterWriteValueInArray_ReadAds[3] := arrCounterWriteValueInArray_ReadAds[3] + 8; arrCounterWriteValueInArray_ReadAds[4] := arrCounterWriteValueInArray_ReadAds[4] + 8;
												arrCounterWriteValueInArray_ReadAds[5] := arrCounterWriteValueInArray_ReadAds[5] + 8; arrCounterWriteValueInArray_ReadAds[6] := arrCounterWriteValueInArray_ReadAds[6] + 8;
													arrCounterWriteValueInArray_ReadAds[7] := arrCounterWriteValueInArray_ReadAds[7] + 8; arrCounterWriteValueInArray_ReadAds[8] := arrCounterWriteValueInArray_ReadAds[8] + 8;			
														IF IsFinite(F_LREAL(unConvertULINT_TO_LREAL_ReadAds.lrValueFloat)) THEN
															IF LEN(LREAL_TO_STRING(unConvertULINT_TO_LREAL_ReadAds.lrValueFloat)) <= 30 THEN 
																IF FIND(LREAL_TO_STRING(unConvertULINT_TO_LREAL_ReadAds.lrValueFloat),'e') = 0 AND FIND(LREAL_TO_STRING(unConvertULINT_TO_LREAL_ReadAds.lrValueFloat),'E') = 0 THEN 
																	sStringFloat_ReadAds := LREAL_TO_STRING(unConvertULINT_TO_LREAL_ReadAds.lrValueFloat);
																		iFindPointFloat_ReadAds := FIND(sStringFloat_ReadAds,'.');
																			sStringFloat_ReadAds := DELETE(sStringFloat_ReadAds,iFindPointFloat_ReadAds,1);
																				iPrecision_ReadAds := LEN(sStringFloat_ReadAds);
																					iPrecision_ReadAds := LIMIT(0,iPrecision_ReadAds,16);
																	IF LEN(LREAL_TO_FMTSTR(unConvertULINT_TO_LREAL_ReadAds.lrValueFloat,iPrecision_ReadAds,TRUE)) <= 30 THEN
																		//Check if the output from Function LREAL_TO_FMTSTR is ok 
																		IF LREAL_TO_FMTSTR(unConvertULINT_TO_LREAL_ReadAds.lrValueFloat,iPrecision_ReadAds,TRUE) <> '#INF' AND LREAL_TO_FMTSTR(unConvertULINT_TO_LREAL_ReadAds.lrValueFloat,iPrecision_ReadAds,TRUE) <> '-#INF' AND
																			LREAL_TO_FMTSTR(unConvertULINT_TO_LREAL_ReadAds.lrValueFloat,iPrecision_ReadAds,TRUE) <> '#QNAN' AND LREAL_TO_FMTSTR(unConvertULINT_TO_LREAL_ReadAds.lrValueFloat,iPrecision_ReadAds,TRUE) <> '-#QNAN' AND
																				LREAL_TO_FMTSTR(unConvertULINT_TO_LREAL_ReadAds.lrValueFloat,iPrecision_ReadAds,TRUE) <> '#OVF' AND LREAL_TO_FMTSTR(unConvertULINT_TO_LREAL_ReadAds.lrValueFloat,iPrecision_ReadAds,TRUE) <> '-#OVF' THEN
																					stADSRead_ReadAds[udiActiveNumberOfSymbol_ReadAds].arrValue[uiLPWriteValueByArray_ReadAds] := LREAL_TO_FMTSTR(unConvertULINT_TO_LREAL_ReadAds.lrValueFloat,iPrecision_ReadAds,TRUE); 
																		ELSE
																			iState_ReadAds := 200;
																				uiInternError_ReadAds := 1;
																		END_IF
																	ELSE
																		//Check if the output from Function LREAL_TO_FMTSTR is ok 
																		IF MID(LREAL_TO_FMTSTR(unConvertULINT_TO_LREAL_ReadAds.lrValueFloat,iPrecision_ReadAds,TRUE),30,1) <> '#INF' AND MID(LREAL_TO_FMTSTR(unConvertULINT_TO_LREAL_ReadAds.lrValueFloat,iPrecision_ReadAds,TRUE),30,1) <> '-#INF' AND
																			MID(LREAL_TO_FMTSTR(unConvertULINT_TO_LREAL_ReadAds.lrValueFloat,iPrecision_ReadAds,TRUE),30,1) <> '#QNAN' AND MID(LREAL_TO_FMTSTR(unConvertULINT_TO_LREAL_ReadAds.lrValueFloat,iPrecision_ReadAds,TRUE),30,1) <> '-#QNAN' AND
																				MID(LREAL_TO_FMTSTR(unConvertULINT_TO_LREAL_ReadAds.lrValueFloat,iPrecision_ReadAds,TRUE),30,1) <> '#OVF' AND MID(LREAL_TO_FMTSTR(unConvertULINT_TO_LREAL_ReadAds.lrValueFloat,iPrecision_ReadAds,TRUE),30,1) <> '-#OVF' THEN
																					stADSRead_ReadAds[udiActiveNumberOfSymbol_ReadAds].arrValue[uiLPWriteValueByArray_ReadAds] := MID(LREAL_TO_FMTSTR(unConvertULINT_TO_LREAL_ReadAds.lrValueFloat,iPrecision_ReadAds,TRUE),30,1);
																		ELSE
																			iState_ReadAds := 200;
																				uiInternError_ReadAds := 1;
																		END_IF 
																	END_IF
																ELSE
																	stADSRead_ReadAds[udiActiveNumberOfSymbol_ReadAds].arrValue[uiLPWriteValueByArray_ReadAds] := LREAL_TO_STRING(unConvertULINT_TO_LREAL_ReadAds.lrValueFloat);
																END_IF
															ELSE
																iState_ReadAds := 200;
																	uiInternError_ReadAds := 1;
															END_IF
														ELSE
															iState_ReadAds := 200;
																uiInternError_ReadAds := 1;
														END_IF
									END_FOR 
								END_IF
					END_IF
				//ARRAY OF STRING(30)
				IF FIND(Lynus_Standards.GVL_Communicator.arrInterfaceInfoAlVariables[byReadWriteArrayNumber,udiActiveNumberOfSymbol_ReadAds].sSymbolType,'OF STRING(30)') <> 0 THEN
					stADSRead_ReadAds[udiActiveNumberOfSymbol_ReadAds].sFullSymbolName := Lynus_Standards.GVL_Communicator.arrInterfaceInfoAlVariables[byReadWriteArrayNumber,udiActiveNumberOfSymbol_ReadAds].sFullSymbolName;
						stADSRead_ReadAds[udiActiveNumberOfSymbol_ReadAds].arrValue := arrValueDefault_ReadAds;	
							IF Lynus_Standards.GVL_Communicator.arrInterfaceInfoAlVariables[byReadWriteArrayNumber,udiActiveNumberOfSymbol_ReadAds].uiSizeArray <= Lynus_Standards.Constants_Communicator.bySizeOfValueArray THEN
								FOR uiLPWriteValueByArray_ReadAds := 1 TO Lynus_Standards.Constants_Communicator.bySizeOfValueArray BY 1 DO 
									FOR byLPCheckCharactersAfterReadOut_ReadAds := 1 TO 31 BY 1 DO
										uiCounterArrayOfString_ReadAds := uiCounterArrayOfString_ReadAds + 1;
											uiCounterArrayOfString_ReadAds := LIMIT(1,uiCounterArrayOfString_ReadAds,1600);	
												stADSRead_ReadAds[udiActiveNumberOfSymbol_ReadAds].arrValue[uiLPWriteValueByArray_ReadAds] := CONCAT(stADSRead_ReadAds[udiActiveNumberOfSymbol_ReadAds].arrValue[uiLPWriteValueByArray_ReadAds],F_ToCHR(arrValueAfterRead_ReadAds[uiCounterArrayOfString_ReadAds]));
													IF arrValueAfterRead_ReadAds[uiCounterArrayOfString_ReadAds] = 0 AND stADSRead_ReadAds[udiActiveNumberOfSymbol_ReadAds].arrValue[uiLPWriteValueByArray_ReadAds] <> '' THEN	
														uiCounterArrayOfString_ReadAds := 31 * uiLPWriteValueByArray_ReadAds;	    
															EXIT; 
													ELSIF arrValueAfterRead_ReadAds[uiCounterArrayOfString_ReadAds] = 0 AND stADSRead_ReadAds[udiActiveNumberOfSymbol_ReadAds].arrValue[uiLPWriteValueByArray_ReadAds] = '' THEN 
														stADSRead_ReadAds[udiActiveNumberOfSymbol_ReadAds].arrValue[uiLPWriteValueByArray_ReadAds] := '#EMPTY#';
															uiCounterArrayOfString_ReadAds := 31 * uiLPWriteValueByArray_ReadAds;
																EXIT;	
													END_IF 
									END_FOR
								END_FOR 
				END_IF		END_IF
					//ARRAY OF TIME or ARRAY OF TIME OF DAY	
					IF FIND(Lynus_Standards.GVL_Communicator.arrInterfaceInfoAlVariables[byReadWriteArrayNumber,udiActiveNumberOfSymbol_ReadAds].sSymbolType,'OF TIME') <> 0 OR FIND(Lynus_Standards.GVL_Communicator.arrInterfaceInfoAlVariables[byReadWriteArrayNumber,udiActiveNumberOfSymbol_ReadAds].sSymbolType,'OF TIME_OF_DAY') <> 0 THEN
						stADSRead_ReadAds[udiActiveNumberOfSymbol_ReadAds].sFullSymbolName := Lynus_Standards.GVL_Communicator.arrInterfaceInfoAlVariables[byReadWriteArrayNumber,udiActiveNumberOfSymbol_ReadAds].sFullSymbolName;
							stADSRead_ReadAds[udiActiveNumberOfSymbol_ReadAds].arrValue := arrValueDefault_ReadAds;	
								IF Lynus_Standards.GVL_Communicator.arrInterfaceInfoAlVariables[byReadWriteArrayNumber,udiActiveNumberOfSymbol_ReadAds].uiSizeArray <= Lynus_Standards.Constants_Communicator.bySizeOfValueArray THEN  
									FOR uiLPWriteValueByArray_ReadAds := 1 TO Lynus_Standards.GVL_Communicator.arrInterfaceInfoAlVariables[byReadWriteArrayNumber,udiActiveNumberOfSymbol_ReadAds].uiSizeArray BY 1 DO
										arrCounterWriteValueInArray_ReadAds[1] := LIMIT(1,arrCounterWriteValueInArray_ReadAds[1],1600); arrCounterWriteValueInArray_ReadAds[2] := LIMIT(2,arrCounterWriteValueInArray_ReadAds[2],1600);
											arrCounterWriteValueInArray_ReadAds[3] := LIMIT(3,arrCounterWriteValueInArray_ReadAds[3],1600); arrCounterWriteValueInArray_ReadAds[4] := LIMIT(4,arrCounterWriteValueInArray_ReadAds[4],1600);
												stADSRead_ReadAds[udiActiveNumberOfSymbol_ReadAds].arrValue[uiLPWriteValueByArray_ReadAds] := UDINT_TO_STRING(SHL(BYTE_TO_UDINT(arrValueAfterRead_ReadAds[arrCounterWriteValueInArray_ReadAds[4]]),24) + SHL(BYTE_TO_UDINT(arrValueAfterRead_ReadAds[arrCounterWriteValueInArray_ReadAds[3]]),16) + SHL(BYTE_TO_UDINT(arrValueAfterRead_ReadAds[arrCounterWriteValueInArray_ReadAds[2]]),8) + BYTE_TO_UDINT(arrValueAfterRead_ReadAds[arrCounterWriteValueInArray_ReadAds[1]]));
										arrCounterWriteValueInArray_ReadAds[1] := arrCounterWriteValueInArray_ReadAds[1] + 4; arrCounterWriteValueInArray_ReadAds[2] := arrCounterWriteValueInArray_ReadAds[2] + 4;
											arrCounterWriteValueInArray_ReadAds[3] := arrCounterWriteValueInArray_ReadAds[3] + 4; arrCounterWriteValueInArray_ReadAds[4] := arrCounterWriteValueInArray_ReadAds[4] + 4;
									END_FOR 
								END_IF
					END_IF
				//ARRAY OF DATE or ARRAY OF DATE AND TIME
				IF FIND(Lynus_Standards.GVL_Communicator.arrInterfaceInfoAlVariables[byReadWriteArrayNumber,udiActiveNumberOfSymbol_ReadAds].sSymbolType,'OF DATE') <> 0 OR FIND(Lynus_Standards.GVL_Communicator.arrInterfaceInfoAlVariables[byReadWriteArrayNumber,udiActiveNumberOfSymbol_ReadAds].sSymbolType,'OF DATE_AND_TIME') <> 0 THEN
					stADSRead_ReadAds[udiActiveNumberOfSymbol_ReadAds].sFullSymbolName := Lynus_Standards.GVL_Communicator.arrInterfaceInfoAlVariables[byReadWriteArrayNumber,udiActiveNumberOfSymbol_ReadAds].sFullSymbolName;
						stADSRead_ReadAds[udiActiveNumberOfSymbol_ReadAds].arrValue := arrValueDefault_ReadAds;	
							IF Lynus_Standards.GVL_Communicator.arrInterfaceInfoAlVariables[byReadWriteArrayNumber,udiActiveNumberOfSymbol_ReadAds].uiSizeArray <= Lynus_Standards.Constants_Communicator.bySizeOfValueArray THEN  
								FOR uiLPWriteValueByArray_ReadAds := 1 TO Lynus_Standards.GVL_Communicator.arrInterfaceInfoAlVariables[byReadWriteArrayNumber,udiActiveNumberOfSymbol_ReadAds].uiSizeArray BY 1 DO
									arrCounterWriteValueInArray_ReadAds[1] := LIMIT(1,arrCounterWriteValueInArray_ReadAds[1],1600); arrCounterWriteValueInArray_ReadAds[2] := LIMIT(2,arrCounterWriteValueInArray_ReadAds[2],1600);
										arrCounterWriteValueInArray_ReadAds[3] := LIMIT(3,arrCounterWriteValueInArray_ReadAds[3],1600); arrCounterWriteValueInArray_ReadAds[4] := LIMIT(4,arrCounterWriteValueInArray_ReadAds[4],1600);
											uliValueDateTime_ReadAds := SHL(BYTE_TO_UDINT(arrValueAfterRead_ReadAds[arrCounterWriteValueInArray_ReadAds[4]]),24) + SHL(BYTE_TO_UDINT(arrValueAfterRead_ReadAds[arrCounterWriteValueInArray_ReadAds[3]]),16) + SHL(BYTE_TO_UDINT(arrValueAfterRead_ReadAds[arrCounterWriteValueInArray_ReadAds[2]]),8) + BYTE_TO_UDINT(arrValueAfterRead_ReadAds[arrCounterWriteValueInArray_ReadAds[1]]);
												uliValueDateTime_ReadAds := uliValueDateTime_ReadAds * 1000;	
													stADSRead_ReadAds[udiActiveNumberOfSymbol_ReadAds].arrValue[uiLPWriteValueByArray_ReadAds] := ULINT_TO_STRING(uliValueDateTime_ReadAds); 
									arrCounterWriteValueInArray_ReadAds[1] := arrCounterWriteValueInArray_ReadAds[1] + 4; arrCounterWriteValueInArray_ReadAds[2] := arrCounterWriteValueInArray_ReadAds[2] + 4;
										arrCounterWriteValueInArray_ReadAds[3] := arrCounterWriteValueInArray_ReadAds[3] + 4; arrCounterWriteValueInArray_ReadAds[4] := arrCounterWriteValueInArray_ReadAds[4] + 4;
								END_FOR 
							END_IF
				END_IF
					
			IF Lynus_Standards.GVL_Communicator.arrInterfaceInfoAlVariables[byReadWriteArrayNumber,udiActiveNumberOfSymbol_ReadAds].uiSizeArray <= Lynus_Standards.Constants_Communicator.bySizeOfValueArray AND iState_ReadAds = 5 THEN 
				arrCounterWriteValueInArray_ReadAds[1] := 0; arrCounterWriteValueInArray_ReadAds[2] := 0; arrCounterWriteValueInArray_ReadAds[3] := 0; 
					arrCounterWriteValueInArray_ReadAds[4] := 0; arrCounterWriteValueInArray_ReadAds[5] := 0; arrCounterWriteValueInArray_ReadAds[6] := 0; 
						arrCounterWriteValueInArray_ReadAds[7] := 0; arrCounterWriteValueInArray_ReadAds[8] := 0;
							uiCounterArrayOfString_ReadAds := 0;
								sStringFloat_ReadAds := ''; iFindPointFloat_ReadAds := 0; iPrecision_ReadAds := 0;
									iState_ReadAds := 6;
			 END_IF			
			
				IF timTimout_ReadAds.Q THEN iState_ReadAds := 200; END_IF
		
		ELSE
			IF udiActiveNumberOfSymbol_ReadAds < Lynus_Standards.GVL_Communicator.arrCounterVariableInArray[byReadWriteArrayNumber] AND udiNumberInProgress_ReadAds < udiNumberSizeValues_ReadAds THEN iState_ReadAds := -4; udiNumberInProgress_ReadAds := udiNumberInProgress_ReadAds + 1; END_IF
			IF (udiNumberInProgress_ReadAds >= udiNumberSizeValues_ReadAds AND iState_ReadAds = 5) THEN iState_ReadAds := -8; udiNumberInProgress_ReadAds := 0; END_IF
			IF udiActiveNumberOfSymbol_ReadAds >= Lynus_Standards.GVL_Communicator.arrCounterVariableInArray[byReadWriteArrayNumber] THEN iState_ReadAds := -8; udiActiveNumberOfSymbol_ReadAds := 0; udiNumberInProgress_ReadAds := 0; udiRestValueSymbolRead_ReadAds := 0; END_IF 
				//Timeout
				IF timTimout_ReadAds.Q THEN iState_ReadAds := 200; END_IF
		END_IF
	
	6://Check if the symbol exist
		byCounterWaitInStep_ReadAds := byCounterWaitInStep_ReadAds + 1;
			byCounterWaitInStep_ReadAds := LIMIT(1,byCounterWaitInStep_ReadAds,2);	
	
		IF byCounterWaitInStep_ReadAds = 1 THEN
			FOR udiLPCheckReadArrays_ReadAds := 1 TO udiNumberLoopHalf_ReadAds BY 1 DO
				IF stADSReadNew_ReadAds[udiLPCheckReadArrays_ReadAds].sFullSymbolName = Lynus_Standards.GVL_Communicator.arrInterfaceInfoAlVariables[byReadWriteArrayNumber,udiActiveNumberOfSymbol_ReadAds].sFullSymbolName THEN 
					iState_ReadAds := 7;																				//Symbol exist in the read array
				END_IF
			END_FOR
		END_IF
			IF byCounterWaitInStep_ReadAds = 2 AND udiNumberLoopFull_ReadAds <> udiNumberLoopHalf_ReadAds THEN
				FOR udiLPCheckReadArrays_ReadAds := (udiNumberLoopHalf_ReadAds + 1) TO udiNumberLoopFull_ReadAds BY 1 DO
					IF stADSReadNew_ReadAds[udiLPCheckReadArrays_ReadAds].sFullSymbolName = Lynus_Standards.GVL_Communicator.arrInterfaceInfoAlVariables[byReadWriteArrayNumber,udiActiveNumberOfSymbol_ReadAds].sFullSymbolName THEN 
						iState_ReadAds := 7;																			//Symbol exist in the read array
					END_IF
				END_FOR
			END_IF
		
				IF byCounterWaitInStep_ReadAds >= 2 AND iState_ReadAds = 6 THEN iState_ReadAds := 9; END_IF 			//Symbol not exist	
				
			//Timeout
			IF timTimout_ReadAds.Q THEN iState_ReadAds := 200; END_IF		
				
	7://Check if the value has changed
		byCounterWaitInStep_ReadAds := 0;
			bValueIsTheSame_ReadAds := FALSE;	
		
		FOR byLPCheckValueChange_ReadAds := 1 TO Lynus_Standards.Constants_Communicator.bySizeOfValueArray BY 1 DO
			IF stADSRead_ReadAds[udiActiveNumberOfSymbol_ReadAds].arrValue[byLPCheckValueChange_ReadAds] <> stADSReadNew_ReadAds[udiActiveNumberOfSymbol_ReadAds].arrValue[byLPCheckValueChange_ReadAds] THEN
				iState_ReadAds := 8;																																				//Value has changed
			ELSE		
				IF iState_ReadAds = 7 AND byLPCheckValueChange_ReadAds >= Lynus_Standards.Constants_Communicator.bySizeOfValueArray THEN iState_ReadAds := 10; bValueIsTheSame_ReadAds := TRUE; END_IF		//Value is the same
			END_IF 
		END_FOR	
		
			//Timeout
			IF timTimout_ReadAds.Q THEN iState_ReadAds := 200; END_IF	
		
	8://Symbol exist and Value has changed
		byCounterWaitInStep_ReadAds := byCounterWaitInStep_ReadAds + 1;
			byCounterWaitInStep_ReadAds := LIMIT(1,byCounterWaitInStep_ReadAds,2);
	
		IF byCounterWaitInStep_ReadAds = 1 THEN 
			FOR udiLPCheckReadArrays_ReadAds := 1 TO udiNumberLoopHalf_ReadAds BY 1 DO
				IF stADSRead_ReadAds[udiLPCheckReadArrays_ReadAds].sFullSymbolName = stADSReadNew_ReadAds[udiLPCheckReadArrays_ReadAds].sFullSymbolName THEN
					stADSReadNew_ReadAds[udiLPCheckReadArrays_ReadAds].arrValue := stADSRead_ReadAds[udiLPCheckReadArrays_ReadAds].arrValue;
				END_IF
			END_FOR
		END_IF	
			IF byCounterWaitInStep_ReadAds = 2 AND udiNumberLoopFull_ReadAds <> udiNumberLoopHalf_ReadAds THEN 
				FOR udiLPCheckReadArrays_ReadAds := (udiNumberLoopHalf_ReadAds + 1) TO udiNumberLoopFull_ReadAds BY 1 DO
					IF stADSRead_ReadAds[udiLPCheckReadArrays_ReadAds].sFullSymbolName = stADSReadNew_ReadAds[udiLPCheckReadArrays_ReadAds].sFullSymbolName THEN
						stADSReadNew_ReadAds[udiLPCheckReadArrays_ReadAds].arrValue := stADSRead_ReadAds[udiLPCheckReadArrays_ReadAds].arrValue;	
					END_IF
				END_FOR
			END_IF 
		
				IF byCounterWaitInStep_ReadAds >= 2 THEN iState_ReadAds := 10; END_IF			
		
			//Timeout
			IF timTimout_ReadAds.Q THEN iState_ReadAds := 200; END_IF
		
	9://Copy the new symbol in the array
		byCounterWaitInStep_ReadAds := 0;
			stADSReadNew_ReadAds := stADSRead_ReadAds;
				iState_ReadAds := 10;
			
	10://Write in Buffer if the send bus is busy or send a messege if the buffer is not empty
		byCounterWaitInStep_ReadAds := 0;
	
		IF NOT Lynus_Standards.GVL_Communicator.arrInterfaceInfoValueSendTo[byReadWriteArrayNumber].bBusy THEN	
			Lynus_Standards.GVL_Communicator.arrInterfaceInfoValueSendTo[byReadWriteArrayNumber].arrValue := arrValueDefault_ReadAds; 						//Clear send Interface if it is no message to send
				Lynus_Standards.GVL_Communicator.arrInterfaceInfoValueSendTo[byReadWriteArrayNumber].sSymbolUnit := ''; 
					Lynus_Standards.GVL_Communicator.arrInterfaceInfoValueSendTo[byReadWriteArrayNumber].sFullSymbolName := '';
						Lynus_Standards.GVL_Communicator.arrInterfaceInfoValueSendTo[byReadWriteArrayNumber].sSymbolType := '';
							IF fbBuffer_ReadAds.nCount > 0 THEN							
								iState_ReadAds := 11;														//Send a new messege from the buffer
							END_IF																			
		END_IF
			IF ((Lynus_Standards.GVL_Communicator.arrInterfaceInfoValueSendTo[byReadWriteArrayNumber].bBusy OR fbBuffer_ReadAds.nCount = 0) AND NOT bValueIsTheSame_ReadAds) THEN
				iState_ReadAds := 20;																		//Insert a new value in the buffer if the send bus is busy or no value is stored in the buffer
			ELSE
				IF iState_ReadAds = 10 THEN 																						
					iState_ReadAds := 100;																	//Value is the same
				END_IF																						
			END_IF
		
			//Timeout
			IF timTimout_ReadAds.Q THEN iState_ReadAds := 200; END_IF
	
	11://Read out a Value from the buffer for sending
		IF udiCounterReadBuffer_New_ReadAds <> fbBuffer_ReadAds.nCount AND fbBuffer_ReadAds.bOk THEN
			udiCounterReadBuffer_New_ReadAds := fbBuffer_ReadAds.nCount;
				IF fbBuffer_ReadAds.cbReturn <= 2000 THEN 
					FOR udiLPCheckReadBuffer_ReadAds := 1 TO fbBuffer_ReadAds.cbReturn BY 1 DO	
						IF byCounterValueReadOut_ReadAds = 0 AND arrBufferRead_ReadAds[udiLPCheckReadBuffer_ReadAds] <> 59 THEN sSymbolNameOutFromBuffer_ReadAds := CONCAT(sSymbolNameOutFromBuffer_ReadAds,F_ToCHR(arrBufferRead_ReadAds[udiLPCheckReadBuffer_ReadAds])); END_IF 
							IF arrBufferRead_ReadAds[udiLPCheckReadBuffer_ReadAds] = 59 THEN byCounterValueReadOut_ReadAds := byCounterValueReadOut_ReadAds + 1; END_IF
								byCounterValueReadOut_ReadAds := LIMIT(0,byCounterValueReadOut_ReadAds,Lynus_Standards.Constants_Communicator.bySizeOfValueArray);
									IF byCounterValueReadOut_ReadAds >= 1 AND arrBufferRead_ReadAds[udiLPCheckReadBuffer_ReadAds] <> 59 AND arrBufferRead_ReadAds[udiLPCheckReadBuffer_ReadAds] <> 0 THEN 
										arrValueOutFromBuffer_ReadAds[byCounterValueReadOut_ReadAds] := CONCAT(arrValueOutFromBuffer_ReadAds[byCounterValueReadOut_ReadAds],F_ToCHR(arrBufferRead_ReadAds[udiLPCheckReadBuffer_ReadAds])); 
									END_IF    	
					END_FOR				 
						IF arrBufferRead_ReadAds[udiLPCheckReadBuffer_ReadAds] = 0 THEN iState_ReadAds := 12; byCounterValueReadOut_ReadAds := 0; END_IF
				END_IF
		END_IF
		
			IF timTimout_ReadAds.Q THEN iState_ReadAds := 200; END_IF
	
	12://Write the Date on interface and start the sending
		byCounterWaitInStep_ReadAds := byCounterWaitInStep_ReadAds + 1;
			byCounterWaitInStep_ReadAds := LIMIT(1,byCounterWaitInStep_ReadAds,2);
	
		IF byCounterWaitInStep_ReadAds = 1 THEN 
			FOR udiLPCheckVarInfoBeforSending_ReadAds := 1 TO udiNumberLoopHalf_ReadAds BY 1 DO
				IF Lynus_Standards.GVL_Communicator.arrInterfaceInfoAlVariables[byReadWriteArrayNumber,udiLPCheckVarInfoBeforSending_ReadAds].sFullSymbolName = sSymbolNameOutFromBuffer_ReadAds THEN
					Lynus_Standards.GVL_Communicator.arrInterfaceInfoValueSendTo[byReadWriteArrayNumber].sFullSymbolName := sSymbolNameOutFromBuffer_ReadAds;
						Lynus_Standards.GVL_Communicator.arrInterfaceInfoValueSendTo[byReadWriteArrayNumber].sSymbolUnit := Lynus_Standards.GVL_Communicator.arrInterfaceInfoAlVariables[byReadWriteArrayNumber,udiLPCheckVarInfoBeforSending_ReadAds].sSymbolUnit;
							Lynus_Standards.GVL_Communicator.arrInterfaceInfoValueSendTo[byReadWriteArrayNumber].sSymbolType := Lynus_Standards.GVL_Communicator.arrInterfaceInfoAlVariables[byReadWriteArrayNumber,udiLPCheckVarInfoBeforSending_ReadAds].sSymbolType;
								Lynus_Standards.GVL_Communicator.arrInterfaceInfoValueSendTo[byReadWriteArrayNumber].arrValue := arrValueOutFromBuffer_ReadAds;
									Lynus_Standards.GVL_Communicator.arrInterfaceInfoValueSendTo[byReadWriteArrayNumber].bBusy := TRUE;
										iState_ReadAds := 13;
											EXIT;	
				END_IF 		 	   	
			END_FOR 	
		END_IF
			IF byCounterWaitInStep_ReadAds = 2 AND udiNumberLoopFull_ReadAds <> udiNumberLoopHalf_ReadAds THEN 
				FOR udiLPCheckVarInfoBeforSending_ReadAds := (udiNumberLoopHalf_ReadAds + 1) TO udiNumberLoopFull_ReadAds BY 1 DO
					IF Lynus_Standards.GVL_Communicator.arrInterfaceInfoAlVariables[byReadWriteArrayNumber,udiLPCheckVarInfoBeforSending_ReadAds].sFullSymbolName = sSymbolNameOutFromBuffer_ReadAds THEN
						Lynus_Standards.GVL_Communicator.arrInterfaceInfoValueSendTo[byReadWriteArrayNumber].sFullSymbolName := sSymbolNameOutFromBuffer_ReadAds;
							Lynus_Standards.GVL_Communicator.arrInterfaceInfoValueSendTo[byReadWriteArrayNumber].sSymbolUnit := Lynus_Standards.GVL_Communicator.arrInterfaceInfoAlVariables[byReadWriteArrayNumber,udiLPCheckVarInfoBeforSending_ReadAds].sSymbolUnit;
								Lynus_Standards.GVL_Communicator.arrInterfaceInfoValueSendTo[byReadWriteArrayNumber].sSymbolType := Lynus_Standards.GVL_Communicator.arrInterfaceInfoAlVariables[byReadWriteArrayNumber,udiLPCheckVarInfoBeforSending_ReadAds].sSymbolType;
									Lynus_Standards.GVL_Communicator.arrInterfaceInfoValueSendTo[byReadWriteArrayNumber].arrValue := arrValueOutFromBuffer_ReadAds;
										Lynus_Standards.GVL_Communicator.arrInterfaceInfoValueSendTo[byReadWriteArrayNumber].bBusy := TRUE;
											iState_ReadAds := 13;
												EXIT;	
					END_IF 		 	   	
				END_FOR 	
			END_IF
		
			IF timTimout_ReadAds.Q THEN iState_ReadAds := 200; END_IF
			
	13://Clear Read Buffer (conserve resources because the code must also work for small plc's)
		byCounterWaitInStep_ReadAds := 0;
			sSymbolNameOutFromBuffer_ReadAds := '';
				MEMCPY(ADR(arrBufferRead_ReadAds),ADR(arrBufferWriteReadDefault_ReadAds),SIZEOF(arrBufferRead_ReadAds));
					arrValueOutFromBuffer_ReadAds := arrValueDefault_ReadAds;
		
			iState_ReadAds := 10;
			
	20://Dim size from the values and symbol name befor can saving in buffer
		uiNumberValueSymbolSize_ReadAds := 0;
			byNumberOfValues_ReadAds_ReadAds := 0;
				byLenghSymbolName_ReadAds := 0;
		FOR byLPDimValueNumberASize_ReadAds := 1 TO Lynus_Standards.Constants_Communicator.bySizeOfValueArray BY 1 DO
			uiNumberValueSymbolSize_ReadAds := uiNumberValueSymbolSize_ReadAds + INT_TO_UINT(LEN(stADSReadNew_ReadAds[udiActiveNumberOfSymbol_ReadAds].arrValue[byLPDimValueNumberASize_ReadAds]));
				IF stADSReadNew_ReadAds[udiActiveNumberOfSymbol_ReadAds].arrValue[byLPDimValueNumberASize_ReadAds] <> '' THEN uiNumberValueSymbolSize_ReadAds := uiNumberValueSymbolSize_ReadAds + 1; END_IF 	
					IF stADSReadNew_ReadAds[udiActiveNumberOfSymbol_ReadAds].arrValue[byLPDimValueNumberASize_ReadAds] <> '' THEN byNumberOfValues_ReadAds_ReadAds := byNumberOfValues_ReadAds_ReadAds + 1; END_IF	
		END_FOR 	
			byLenghSymbolName_ReadAds := INT_TO_BYTE(LEN(stADSReadNew_ReadAds[udiActiveNumberOfSymbol_ReadAds].sFullSymbolName));
				uiNumberValueSymbolSize_ReadAds := uiNumberValueSymbolSize_ReadAds + byLenghSymbolName_ReadAds + 1;
		
			IF byNumberOfValues_ReadAds_ReadAds <= Lynus_Standards.Constants_Communicator.bySizeOfValueArray THEN
				FOR byLPDimLenghValues_ReadAds := 1 TO byNumberOfValues_ReadAds_ReadAds BY 1 DO
					arrLenghEachValue_ReadAds[byLPDimLenghValues_ReadAds] := INT_TO_BYTE(LEN(stADSReadNew_ReadAds[udiActiveNumberOfSymbol_ReadAds].arrValue[byLPDimLenghValues_ReadAds]));	
				END_FOR 
			END_IF
	
		IF byNumberOfValues_ReadAds_ReadAds <= Lynus_Standards.Constants_Communicator.bySizeOfValueArray AND byNumberOfValues_ReadAds_ReadAds >= 1 AND uiNumberValueSymbolSize_ReadAds <> 0 THEN iState_ReadAds := 21; END_IF
		
			IF timTimout_ReadAds.Q THEN iState_ReadAds := 200; END_IF
			
	21://String to Ascii Symbol Name and values
		IF byLenghSymbolName_ReadAds <= 49 THEN
			FOR byLPSymbolNameToAscii_ReadAds := 1 TO byLenghSymbolName_ReadAds BY 1 DO
				arrSymbolName_ReadAds[byLPSymbolNameToAscii_ReadAds] := F_ToASC(MID(stADSReadNew_ReadAds[udiActiveNumberOfSymbol_ReadAds].sFullSymbolName,1,byLPSymbolNameToAscii_ReadAds));
			END_FOR 
		END_IF
			IF byLenghSymbolName_ReadAds < 49 THEN arrSymbolName_ReadAds[byLenghSymbolName_ReadAds + 1] := F_ToASC(';'); END_IF  	
		
		IF byNumberOfValues_ReadAds_ReadAds <= Lynus_Standards.Constants_Communicator.bySizeOfValueArray THEN 
			FOR byLPValueNameToAscii_1_ReadAds := 1 TO byNumberOfValues_ReadAds_ReadAds BY 1 DO
				IF arrLenghEachValue_ReadAds[byLPValueNameToAscii_1_ReadAds] <= 31 THEN 
					FOR byLPValueNameToAscii_2_ReadAds := 1 TO arrLenghEachValue_ReadAds[byLPValueNameToAscii_1_ReadAds] BY 1 DO
						arrValueName_ReadAds[byLPValueNameToAscii_1_ReadAds,byLPValueNameToAscii_2_ReadAds] := F_ToASC(MID(stADSReadNew_ReadAds[udiActiveNumberOfSymbol_ReadAds].arrValue[byLPValueNameToAscii_1_ReadAds],1,byLPValueNameToAscii_2_ReadAds));
					END_FOR
				END_IF
					arrValueName_ReadAds[byLPValueNameToAscii_1_ReadAds,byLPValueNameToAscii_2_ReadAds] := F_ToASC(';'); 			
			END_FOR 
		END_IF 
		
		IF byLenghSymbolName_ReadAds <= 49 AND byNumberOfValues_ReadAds_ReadAds <= Lynus_Standards.Constants_Communicator.bySizeOfValueArray AND arrLenghEachValue_ReadAds[byNumberOfValues_ReadAds_ReadAds] <= 31 THEN iState_ReadAds := 22; END_IF
		
			IF timTimout_ReadAds.Q THEN iState_ReadAds := 200; END_IF	
			
	22://Prepare Write array for Buffer
		IF byLenghSymbolName_ReadAds <= 48 THEN
			FOR uiLPWriteByteValueInArray_ReadAds := 1 TO (byLenghSymbolName_ReadAds + 1) BY 1 DO
				arrBufferWrite_ReadAds[uiLPWriteByteValueInArray_ReadAds] := arrSymbolName_ReadAds[uiLPWriteByteValueInArray_ReadAds];
			END_FOR 
		END_IF
		
		IF byLenghSymbolName_ReadAds <= 48 THEN	iState_ReadAds := 23; END_IF
			
			IF timTimout_ReadAds.Q THEN iState_ReadAds := 200; END_IF
	
	23://Prepare Write array for Buffer
		uiValueForLoopStart_ReadAds := uiLPWriteByteValueInArray_ReadAds;
			byValueInTurn_ReadAds := byValueInTurn_ReadAds + 1;
				byValueInTurn_ReadAds := LIMIT(1,byValueInTurn_ReadAds,Lynus_Standards.Constants_Communicator.bySizeOfValueArray);
					uiValueForLoopStop_ReadAds := arrLenghEachValue_ReadAds[byValueInTurn_ReadAds] + uiValueForLoopStart_ReadAds;
						byCounterValue_ReadAds := 0;
							
							IF uiValueForLoopStart_ReadAds >= 1 AND uiValueForLoopStart_ReadAds <= 2000 AND uiValueForLoopStop_ReadAds >= 1 AND uiValueForLoopStop_ReadAds <= 2000 THEN 
								FOR uiLPWriteByteValueInArray_ReadAds := uiValueForLoopStart_ReadAds TO uiValueForLoopStop_ReadAds BY 1 DO
									byCounterValue_ReadAds :=  byCounterValue_ReadAds + 1;
										byCounterValue_ReadAds := LIMIT(1,byCounterValue_ReadAds,31);	
											arrBufferWrite_ReadAds[uiLPWriteByteValueInArray_ReadAds] := arrValueName_ReadAds[byValueInTurn_ReadAds,byCounterValue_ReadAds];
								END_FOR 
							END_IF
		
		IF byValueInTurn_ReadAds >= byNumberOfValues_ReadAds_ReadAds AND uiValueForLoopStart_ReadAds >= 1 AND uiValueForLoopStart_ReadAds <= 2000 AND uiValueForLoopStop_ReadAds >= 1 AND uiValueForLoopStop_ReadAds <= 2000 THEN 
			iState_ReadAds := 24; 
				uiValueForLoopStart_ReadAds := 0;
					byValueInTurn_ReadAds := 0;
						uiValueForLoopStop_ReadAds := 0;
							byCounterValue_ReadAds := 0;			
		END_IF
			
			IF timTimout_ReadAds.Q THEN iState_ReadAds := 200; END_IF

	24://Write Value in Buffer
		iState_ReadAds := 25; 
				
	25://Check if the new value is stored in the buffer
		IF fbBuffer_ReadAds.bOk AND fbBuffer_ReadAds.nCount <> udiCounterReadBuffer_New_ReadAds THEN udiCounterReadBuffer_New_ReadAds := fbBuffer_ReadAds.nCount; iState_ReadAds := 26; END_IF  	
			
			IF timTimout_ReadAds.Q THEN iState_ReadAds := 200; END_IF
		
	26://Clear the Write Buffer (conserve resources because the code must also work for small plc's)
		MEMCPY(ADR(arrBufferWrite_ReadAds),ADR(arrBufferWriteReadDefault_ReadAds),SIZEOF(arrBufferWrite_ReadAds));
		
			iState_ReadAds := 100;

	100://Check for other variable
		//Next symbol
		IF udiActiveNumberOfSymbol_ReadAds < Lynus_Standards.GVL_Communicator.arrCounterVariableInArray[byReadWriteArrayNumber] AND udiNumberInProgress_ReadAds < udiNumberSizeValues_ReadAds THEN iState_ReadAds := -4; udiNumberInProgress_ReadAds := udiNumberInProgress_ReadAds + 1; END_IF
			//Start with the next 10 Variables
			IF (udiNumberInProgress_ReadAds >= udiNumberSizeValues_ReadAds AND iState_ReadAds = 100) THEN 
				iState_ReadAds := -8; 
					udiNumberInProgress_ReadAds := 0;
			END_IF	
				//Start from New with the first 10 Variables 	
				IF udiActiveNumberOfSymbol_ReadAds >= Lynus_Standards.GVL_Communicator.arrCounterVariableInArray[byReadWriteArrayNumber] THEN
					iState_ReadAds := -8; 
						udiActiveNumberOfSymbol_ReadAds := 0;
							udiNumberInProgress_ReadAds := 0;
								udiRestValueSymbolRead_ReadAds := 0;
						 			bFirstReadCycleDone_ReadAds := TRUE; 
				END_IF			
			
			bError_ReadAds := FALSE;
				uiInternError_ReadAds := 0;
			
			IF timTimout_ReadAds.Q THEN iState_ReadAds := 200; END_IF
				
	200://Error
		bError_ReadAds := TRUE; fbADSREADWRITE_ReadAds.WRTRD := FALSE; bValueIsTheSame_ReadAds := FALSE; 
			udiActiveNumberOfSymbol_ReadAds := 0; byCounterWaitInStep_ReadAds := 0; udiNumberInProgress_ReadAds := 0; udiRestValueSymbolRead_ReadAds := 0;
		
		//Clear the write Buffer befor go to step 0 (conserve resources because the code must also work for small plc's)
		MEMCPY(ADR(arrBufferWrite_ReadAds),ADR(arrBufferWriteReadDefault_ReadAds),SIZEOF(arrBufferWrite_ReadAds));
		
		//Clear the read Buffer befor go to step 0 (conserve resources because the code must also work for small plc's)
		sSymbolNameOutFromBuffer_ReadAds := '';
			MEMCPY(ADR(arrBufferRead_ReadAds),ADR(arrBufferWriteReadDefault_ReadAds),SIZEOF(arrBufferRead_ReadAds));
				arrValueOutFromBuffer_ReadAds := arrValueDefault_ReadAds;
			
		//Count up when an error has occurred
		byErrorCounter_ReadAds := byErrorCounter_ReadAds + 1;		
				
			iState_ReadAds := 300;
	
	300://Wait in Error and clear the rest from the read and write buffer (conserve resources because the code must also work for small plc's)
		byCounterWaitInStep_ReadAds := byCounterWaitInStep_ReadAds + 1;
	
			//Restart new from in Step -8. No Reset from the complete System
			IF byCounterWaitInStep_ReadAds > 10 AND byErrorCounter_ReadAds <= 10 THEN byCounterWaitInStep_ReadAds := 0; iState_ReadAds := -8; END_IF
				//Restart new from in Step -10. Reset from the complete System after to much Errors
				IF byCounterWaitInStep_ReadAds > 10 AND byErrorCounter_ReadAds > 10 THEN 
						byCounterWaitInStep_ReadAds := 0; 
							//Reset Read Steps and start from new
							iState_ReadAds := -10;
								//Reset Write Steps and start from new
								iState_WriteAds := -2;
									byErrorCounter_ReadAds := 0; 
				END_IF
	
END_CASE	

//Resetting the error counter after not being in the error step for 30 min
timResetErrorCounter_ReadAds(IN:= byErrorCounter_ReadAds <> 0, PT:= T#30M, Q=> , ET=> );
	IF timResetErrorCounter_ReadAds.Q THEN byErrorCounter_ReadAds := 0; END_IF 

//Read Out Variable by ADS
fbADSREADWRITE_ReadAds(
	NETID:= fbNedID.AddrString, 
	PORT:= uiPort, 
	IDXGRP:= 16#F080, 
	IDXOFFS:= udiNumberSizeValues_ReadAds, 
	WRITELEN:= , 
	READLEN:= udiSizeReq_ReadAds, 
	SRCADDR:= , 
	DESTADDR:= ADR(arrValueRead_ReadAds), 
	WRTRD:= , 
	TMOUT:= T#5S, 
	BUSY=> , 
	ERR=> , 
	ERRID=> );

FPErrorReadWrite_ReadAds(CLK:= fbADSREADWRITE_ReadAds.ERR, Q=> );	
	
//Buffer Read Value from ADS
FPWriteValueToBufferStep25_ReadAds(CLK:= iState_ReadAds = 24, Q=> );
FPReadValueToBufferStep11_ReadAds(CLK:= iState_ReadAds = 11, Q=> );

IF FPReadValueToBufferStep11_ReadAds.Q THEN fbBuffer_ReadAds.A_RemoveHead(); END_IF
IF FPWriteValueToBufferStep25_ReadAds.Q THEN fbBuffer_ReadAds.A_AddTail(); END_IF

//Reset the Buffer after a Buffer Overflow
IF fbBuffer_ReadAds.nCount <> 0 AND NOT fbBuffer_ReadAds.bOk THEN timResetBuffer_ReadAds.IN := TRUE; ELSE timResetBuffer_ReadAds.IN := FALSE; END_IF
	timResetBuffer_ReadAds(IN:= , PT:= T#40S, Q=> , ET=> );
		IF timResetBuffer_ReadAds.Q THEN fbBuffer_ReadAds.A_Reset(); END_IF

fbBuffer_ReadAds(
	pWrite:= ADR(arrBufferWrite_ReadAds), 
	cbWrite:= uiNumberValueSymbolSize_ReadAds, 
	pRead:= ADR(arrBufferRead_ReadAds), 
	cbRead:= SIZEOF(arrBufferRead_ReadAds), 
	pBuffer:= ADR(arrBufferADSRead_ReadAds), 
	cbBuffer:= SIZEOF(arrBufferADSRead_ReadAds), 
	bOk=> Lynus_Standards.GVL_Communicator.arrInterfaceInfoValueSendTo[byReadWriteArrayNumber].bBufferOK, 
	nCount=> Lynus_Standards.GVL_Communicator.arrInterfaceInfoValueSendTo[byReadWriteArrayNumber].udiCountBuffer, 
	cbSize=> , 
	cbReturn=> );

END_IF
	
//Busy
IF iState_ReadAds >= -8 OR iState_WriteAds >= 0 THEN bBusy := TRUE; ELSE bBusy := FALSE; END_IF
	
//Error
IF (bError_ReadAds AND iState_ReadAds <> - 10 AND iState_ReadAds <> - 9) OR (bError_WriteAds AND iState_WriteAds <> - 1 AND iState_WriteAds <> - 2) THEN fbErrorCodes.bErrorIntern := TRUE; ELSE fbErrorCodes.bErrorIntern := FALSE; END_IF

IF fbADSREADWRITE_ReadAds.ERR OR fbADSREADWRITE_WriteAds.ERR OR fbADSWrite_WriteAds.ERR THEN fbErrorCodes.bErrorADS := TRUE; END_IF

IF fbADSREADWRITE_ReadAds.ERR THEN fbErrorCodes.udiErrorCodeADS := fbADSREADWRITE_ReadAds.ERRID; END_IF
IF fbADSREADWRITE_WriteAds.ERR THEN fbErrorCodes.udiErrorCodeADS := fbADSREADWRITE_WriteAds.ERRID; END_IF
IF fbADSWrite_WriteAds.ERR THEN fbErrorCodes.udiErrorCodeADS := fbADSWrite_WriteAds.ERRID; END_IF

IF NOT fbADSREADWRITE_ReadAds.ERR AND NOT fbADSREADWRITE_ReadAds.BUSY AND NOT
	fbADSREADWRITE_WriteAds.ERR AND NOT fbADSREADWRITE_WriteAds.BUSY AND NOT fbADSWrite_WriteAds.ERR AND NOT fbADSWrite_WriteAds.BUSY THEN 
		fbErrorCodes.bErrorADS := FALSE;
			fbErrorCodes.udiErrorCodeADS := 0; 
END_IF 	     
	
fbErrorCodes(
	bErrorADS:= , 
	bErrorIntern:= , 
	udiErrorCodeADS:= , 
	udiErrorCodesInternRead:= uiInternError_ReadAds, 
	udiErrorCodesInternWrite:= uiInternError_WriteAds, 
	udiErrorCodeADS_Out=> udiErrorCodeOut, 
	bError=> bError, 
	eErrorReadWrite_Out=> eErrorReadWrite_Out);

END_FUNCTION_BLOCK

// ---- FB/FB_ReadWrite_V2.TcPOU
// {attribute 'hide_all_locals'}
FUNCTION_BLOCK FB_ReadWrite_V2
VAR_INPUT
	eUploadType							:eSelectDataUploadType;		//0:NoChange+Intervall 5min 1:NoChange+Intervall 1min 2:Change+noIntervall 3:Change+Intervall 5min 4:Change+Intervall 1min
END_VAR
VAR_OUTPUT
	bBusy													: BOOL;																								//Busy flag
	bError													: BOOL;																								//Error flag
	udiErrorCodeOut											: UDINT;																							//Error ID		
	eErrorReadWrite_Out										: eErrorReadWrite;																					//Enum with Error from the read/write function
END_VAR
VAR
	(*-----------------------------------------------------------------------------------------Other-------------------------------------------------------------------------------------------------------*)
	fbNedID													: FB_GetLocalAmsNetId := (bExecute := TRUE);														//Read net id from PLC	
	fbTaskIndex												: GETCURTASKINDEX;																					//Task Index
	fbErrorCodes											: FB_VarReadWrite_ErrorCodes;																		//Function for error codes
	FPInitSendError											: R_TRIG;																							//Internal rising edge 
	timTimerStart											: TON;																								//Timer to start the ReadWrite (Start one after the other if there are several ReadWrite functions)
	byStaticValueWaitInStep									: BYTE;																								//Static Value for wait in step
	byReadWriteArrayNumber									: BYTE;																								//Read write array in use
	byLPReadWriteArrayNumber								: BYTE;																								//Loop to find out a free number from the array
	uiPort													: UINT;																								//TC port
	udiCycleTime											: UDINT;																							//Cycle Time
	(*-----------------------------------------------------------------------------------------ADS READ-------------------------------------------------------------------------------------------------------*)
	fbADSREADWRITE_ReadAds									: ADSRDWRT;																							//ADS read/write function
	unConvertDWORD_TO_REAL_ReadAds							: ST_UN_FLOAT_CONVERT_DWORD_REAL;																	//Union to convert numbers
	unConvertULINT_TO_LREAL_ReadAds							: ST_UN_FLOAT_CONVERT_ULINT_LREAL;																	//Union to convert numbers
	fbBuffer_ReadAds										: FB_MemRingBuffer;																					//Ringbuffer read
	FPErrorReadWrite_ReadAds								: R_TRIG;																							//Internal rising edge 
	FPWriteValueToBufferStep25_ReadAds						: R_TRIG;																							//Internal rising edge 
	FPReadValueToBufferStep11_ReadAds						: R_TRIG;																							//Internal rising edge 
	timTimout_ReadAds										: TON;																								//Timout timer
	timResetBuffer_ReadAds									: TON;																								//Timer to Reset the Buffer after a Buffer Overflow
	timResetErrorCounter_ReadAds							: TON;																								//Timer to Reset the Error Counter when a longer Time we dont go inside the Error State
	stADSReadDefault_ReadAds								: ARRAY[1..Lynus_Standards.Constants_Communicator.udiArraySizeMarkedSymobls] OF ST_SymbolRead;		//Array with the default Data of al matching variables
	stADSRead_ReadAds										: ARRAY[1..Lynus_Standards.Constants_Communicator.udiArraySizeMarkedSymobls] OF ST_SymbolRead;		//Array with the Data of al matching variables
	stADSReadNew_ReadAds									: ARRAY[1..Lynus_Standards.Constants_Communicator.udiArraySizeMarkedSymobls] OF ST_SymbolRead;		//Array with the Data of al matching variables
	arrInfoValue_Read_Ads									: ARRAY[1..10] OF ST_BlockReadValue;																//Struct with symbol values
	arrValueAfterRead_ReadAds								: ARRAY[1..1600] OF BYTE;																			//Buffer after reat out data
	arrValueAfterReadDefault_ReadAds						: ARRAY[1..1600] OF BYTE;																			//Buffer after reat out data default
	arrValueRead_ReadAds									: ARRAY[1..16000] OF BYTE;																			//Buffer size for read function
	arrSymbolName_ReadAds									: ARRAY[1..49] OF BYTE;																				//Smybol name in single chracters	
	arrSymbolNameDefault_ReadAds							: ARRAY[1..49] OF BYTE;																				//Default Smybol name in single chracters	
	arrValueName_ReadAds									: ARRAY[1..Lynus_Standards.Constants_Communicator.bySizeOfValueArray,1..31] OF BYTE;				//Value name in single chracters	
	arrValueNameDefault_ReadAds								: ARRAY[1..Lynus_Standards.Constants_Communicator.bySizeOfValueArray,1..31] OF BYTE;				//Default Value name in single chracters 	
	arrLenghEachValue_ReadAds								: ARRAY[1..Lynus_Standards.Constants_Communicator.bySizeOfValueArray] OF BYTE; 						//Lengt of each value
	arrLenghEachValueDefault_ReadAds						: ARRAY[1..Lynus_Standards.Constants_Communicator.bySizeOfValueArray] OF BYTE; 						//Default Lengt of each value 	
	arrBufferADSRead_ReadAds								: ARRAY[1..32000] OF BYTE;																			//Buffer read size
	arrBufferRead_ReadAds									: ARRAY[1..2000] OF BYTE;																			//Value read out from send buffer
	arrBufferWrite_ReadAds									: ARRAY[1..2000] OF BYTE;																			//Value to write in buffer
	arrBufferWriteReadDefault_ReadAds						: ARRAY[1..2000] OF BYTE;																			//Default buffer for read and write 
	arrReqValue_ReadAds										: ARRAY[1..10,1..12] OF BYTE;																		//Data for Block Request
	arrBufferReq_ReadAds									: ARRAY[1..120] OF BYTE;																			//Data for Block Request
	arrCounterWriteValueInArray_ReadAds						: ARRAY[1..8] OF UINT;																				//Counter to write the read value if it is a array
	arrValueDefault_ReadAds									: ARRAY[1..Lynus_Standards.Constants_Communicator.bySizeOfValueArray] OF STRING(30);				//Default Value from the Variable
	arrValueOutFromBuffer_ReadAds							: ARRAY[1..Lynus_Standards.Constants_Communicator.bySizeOfValueArray] OF STRING(30);				//Values from read Buffer
	arrCounterValueSymbolReads_ReadAds						: ARRAY[1..10] OF UDINT;																			//Counter to read out symbols
	sSymbolNameOutFromBuffer_ReadAds						: STRING(48);																						//Symbol Name from read Buffer
	bValueIsTheSame_ReadAds									: BOOL;																								//True Symbol has the same value; False Symbol has changed the value
	bError_ReadAds											: BOOL;																								//Error flag
	bFirstReadCycleDone_ReadAds								: BOOL;																								//True if the first read cycle is done. Befor write value is deactivated
	byErrorCounter_ReadAds									: BYTE;																								//Counter entryes in the Error State
	byCounterWaitInStep_ReadAds								: BYTE;																								//Wait counter in statemschine
	byLPDimValueNumberASize_ReadAds							: BYTE;																								//Loop to dim numer of values and the size
	byLPSymbolNameToAscii_ReadAds							: BYTE;																								//Loop to write the symbol name as asci in the array
	byLPValueNameToAscii_1_ReadAds							: BYTE;																								//Loop to write the value name as asci in the array
	byLPValueNameToAscii_2_ReadAds							: BYTE;																								//Loop to write the value name as asci in the array
	byLPDimLenghValues_ReadAds								: BYTE;																								//Loop to dim lengh of the values
	byLPCheckValueChange_ReadAds							: BYTE;																								//Loop to check the value change
	byLPCheckCharactersAfterReadOut_ReadAds					: BYTE;																								//Loop to convert the Byte after read out in Characters
	byLPClearStructs_ReadAds								: BYTE;																								//Loop to clear structs
	byLPFillBufferReq_1_ReadAds								: BYTE;																								//Loop to fill the request buffer
	byLPFillBufferReq_2_ReadAds								: BYTE;																								//Loop to fill the request buffer
	byNumberOfValues_ReadAds_ReadAds						: BYTE;																								//Number of values befor saving in the buffer
	byLenghSymbolName_ReadAds								: BYTE;																								//Size of the symbol name befor saving
	byValueInTurn_ReadAds									: BYTE;																								//Value in turn when filling the write array
	byCounterValue_ReadAds									: BYTE;																								//Value currently being written into the array
	byCounterValueReadOut_ReadAds							: BYTE;																								//Counter to encode the read out Data from buffer
	byCounterBufferReq_ReadAds								: BYTE;																								//Counter to fill the request buffer																					
	iState_ReadAds											: INT := -2;																						//Statemaschine for ADS Read
	iFindPointFloat_ReadAds									: INT;																								//Variable to find the point in the float value
	iPrecision_ReadAds										: INT;																								//Precision for float value
	uiNumberValueSymbolSize_ReadAds							: UINT;																								//Size of the complete charachters befror store in the buffer
	uiLPWriteValueByArray_ReadAds							: UINT;																								//Loop to write the values from the read ads data in the array of values
	uiLPWriteByteValueInArray_ReadAds						: UINT;																								//Loop to write the values in the write array
	uiValueForLoopStart_ReadAds								: UINT;																								//Value start for loop write value in write array
	uiValueForLoopStop_ReadAds								: UINT;																								//Value stop for loop write value in write array
	uiInternError_ReadAds									: UINT;																								//Intern Error Code Read ads
	uiCounterArrayOfString_ReadAds							: UINT;																								//Counter to encode the array form the read value
	uiCounterCopyValueFromReqBuffer_ReadAds					: UINT;																								//Conter to copy the value from big intern buffer to small buffer
	udiLPCheckReadArrays_ReadAds							: UDINT;																							//Loop to check the read array for name and value
	udiLPCheckReadBuffer_ReadAds							: UDINT;																							//Loop to check the symbols in the read buffer
	udiLPCheckVarInfoBeforSending_ReadAds					: UDINT;																							//Loop to check the var info befor sending
	udiLPCheckErrorAfterReadReq_ReadAds						: UDINT;																							//Loop to check Error after read out
	udiLPCopyValueFromReqBuffer_ReadAds						: UDINT;																							//Loop to copy the values from request buffer
	udiActiveNumberOfSymbol_ReadAds							: UDINT;																							//Number of the Varaibele that is currently being read out
	udiCounterReadBuffer_New_ReadAds						: UDINT;																							//Counter to check if the new value is stored in the buffer
	udiNumberLoopFull_ReadAds								: UDINT;																							//Number of the max Loop (dependet from max symbols in plc)
	udiNumberLoopHalf_ReadAds								: UDINT;																							//Number of the max Loop /2 (dependet from max symbols in plc)
	udiStartValueSymbolsRead_ReadAds						: UDINT;																							//Start value to read the symbols
	udiStopValueSymbolsRead_ReadAds							: UDINT;																							//Stop value to read the symbols
	udiRestValueSymbolRead_ReadAds							: UDINT;																							//Remain from the symbols not yet read 
	udiSizeReq_ReadAds										: UDINT;																							//Size from read request
	udiNumberSizeValues_ReadAds								: UDINT;																							//Number of symbols
	udiStartValueReadOutReqBuffer_AdsRead					: UDINT;																							//Start value to read out from the big buffer																						
	udiStopValueReadOutReqBuffer_AdsRead					: UDINT;																							//Stop value to read out from the big buffer
	udiNumberInProgress_ReadAds								: UDINT;																							//Number in prgogress from the 10 read out values
	uliValueDateTime_ReadAds								: ULINT;																							//Value Date and time after read out in milliseconds
	sStringFloat_ReadAds									: STRING(510);																						//String to check the float value
	(*-----------------------------------------------------------------------------------------ADS WRITE-------------------------------------------------------------------------------------------------------*)
	fbADSREADWRITE_WriteAds									: ADSRDWRT;																							//ADS read/write function
	fbADSWrite_WriteAds										: ADSWRITE;																							//ADS write function
	FPErrorWrite_WriteAds									: R_TRIG;																							//Internal rising edge 
	FPErrorReadWrite_WriteAds								: R_TRIG;																							//Internal rising edge 
	timTimout_WriteAds										: TON;																								//Timout timer
	unConvertDWORD_TO_REAL_WriteAds							: ST_UN_FLOAT_CONVERT_DWORD_REAL;																	//Union to convert numbers
	unConvertULINT_TO_LREAL_WriteAds						: ST_UN_FLOAT_CONVERT_ULINT_LREAL;																	//Union to convert numbers
	arrBufferWriteDefault_WriteAds							: ARRAY[1..2000] OF BYTE;																			//Default Value to write ofer ads
	arrBufferWrite_WriteAds									: ARRAY[1..2000] OF BYTE;																			//Value to write ofer ads
	arrCounterWriteValueInArray_WriteAds					: ARRAY[1..8] OF UINT;																				//Counter to write the received value in the array
	arrValueDefault											: ARRAY[1..Lynus_Standards.Constants_Communicator.bySizeOfValueArray] OF STRING(30);				//Default values
	bError_WriteAds											: BOOL;																								//Error flag
	bValueValid_WriteAds									: BOOL;																								//True if the received value for write over ads is valid
	byCounterWaitInStep_WriteAds							: BYTE;																								//Wait counter in statemschine
	byCounterEncodeString_WriteAds							: BYTE;																								//Counter to encode the received String befor write ofer ads
	byCounterReceivedValueOK_WriteAds						: BYTE;																								//Counter for fill write array
	byLPEncodeReceivedString_WriteAds						: BYTE;																								//Loop to encode the received string
	iState_WriteAds											: INT := -2;																						//State maschine to write ADS
	uiInternError_WriteAds									: UINT;																								//Intern Error Code Write ads
	uiSizeToWrite_WriteAds									: UINT;																								//Size from the value befor write oder ads
	uiLPWriteValueFromArray_WriteAds						: UINT;																								//Loop to write the values from received messege in the write buffer
	uiCounterEncodeString_WriteAds							: UINT;																								//Counter to encode the received String befor write ofer ads
	uiWaitBySymbolString_WriteAds							: UINT;																								//If array is located, extend wait step due to ads write access
	udiDate_WriteAds										: UDINT;																							//Received Date or Daten and time
	udiLPWriteInReadArrayForCheck_WriteADS					: UDINT;																							//Loop to write the new Value in the read array. If the value not can write with success, the old read value is pushing in next step to the cloud 
	dwVarHndl_WriteAds										: DWORD;																							//Handle to read or write on the variable
	uliDate_WriteAds										: ULINT;																							//Received Date or Daten and time
	rRealValueCheckBeforWrite_WriteAds						: REAL;																								//Need to check the Real Value befror write in Buffer
	lrRealValueCheckBeforWrite_WriteAds						: LREAL;																							//Need to check the lReal Value befror write in Buffer
(*------------------------------------------------interval sending -----------------------------------------*)	
	m_EnableChange_upload	:BOOL;
	m_EnableInterval		:BOOL;
	time_Interval			:TIME:=T#1M;

	timer_Interval											: Ton;
	m_TriggerIntervalSend										: BOOL;
END_VAR

//Creator : Stefan Lackner
//Company : EfficientIO
//Date : 12.10.2022
//Version : 1.0.0.2

//With this function its possible to read and write data from the symbols that were first found with the info Var find function
//The read function from the values of the symbols is cyclically, because directly on the plc is not possible to work with notifications 
//The read function always reads 10 variables at the same time. (Block Mode)
//At the beginning all variables are saved.
//After that, the whole direction works based on the buffer event, i.e. the value is only written to the buffer if it also changes
//If the send interface is free, the messages are sent from the buffer. Typ FIFO
//The function only starts when the scan module has been successfully completed and a connection to the cloud has been established.
//If there are several read and write functions on the PLC, then divide up the number of symbols. (Max 10 read write functions on 1 plc)
// Changes in Version 1.0.0.2
// added Input 	eUploadType		:eSelectDataUploadType; and the necessary functions
// 




//Define Array Number for this function
IF Lynus_Standards.GVL_Communicator.bBusyInfoAlVariables OR Lynus_Standards.GVL_Communicator.bErrorInfoAlVariables OR NOT Lynus_Standards.GVL_Communicator.bInfoAlVariablesOK THEN 
	byReadWriteArrayNumber := 0; 
		iState_ReadAds := -10;
			iState_WriteAds := -2;
				timTimerStart.IN := FALSE; 	
END_IF  

IF byReadWriteArrayNumber = 0 AND NOT Lynus_Standards.GVL_Communicator.bBusyInfoAlVariables AND Lynus_Standards.GVL_Communicator.bInfoAlVariablesOK THEN
	FOR byLPReadWriteArrayNumber := 1 TO 10 BY 1 DO
		IF NOT Lynus_Standards.GVL_Communicator.arrReadWriteArrayNumberInUse[byLPReadWriteArrayNumber] THEN
			byReadWriteArrayNumber := Lynus_Standards.GVL_Communicator.arrReadWriteArrayNumber[byLPReadWriteArrayNumber];
				Lynus_Standards.GVL_Communicator.arrReadWriteArrayNumberInUse[byLPReadWriteArrayNumber] := TRUE;
					timTimerStart.IN := TRUE; 
						EXIT;
		END_IF	 	 
	END_FOR
END_IF

timTimerStart(IN:= , PT:= T#500MS * byReadWriteArrayNumber, Q=> , ET=> );

//Start from here with the general code. All of the code is inside this IF instruction 
IF byReadWriteArrayNumber <> 0 AND timTimerStart.Q THEN

byReadWriteArrayNumber := LIMIT(1,byReadWriteArrayNumber,10);

//TC3 Port
uiPort := TwinCAT_SystemInfoVarList._AppInfo.AdsPort;

//AMS Net ID
fbNedID();
	IF (NOT fbNedID.bBusy) AND NOT fbNedID.bError THEN fbNedID.bExecute := FALSE; END_IF

//TaskIndex
fbTaskIndex(index=> );
	udiCycleTime := TwinCAT_SystemInfoVarList._TaskInfo[fbTaskIndex.index].CycleTime / 10000;	
	
//Wait in Step min 3 x Cycle Time for ADS Response
byStaticValueWaitInStep := STRING_TO_BYTE(LREAL_TO_FMTSTR((UDINT_TO_LREAL(udiCycleTime) / 10) * 3,0,FALSE)); 
	byStaticValueWaitInStep := LIMIT(3,byStaticValueWaitInStep,30);	
 
//Timeout
IF iState_ReadAds <> -8 AND iState_ReadAds <> -9 AND iState_ReadAds <> -4 THEN timTimout_ReadAds.IN := TRUE; ELSE timTimout_ReadAds.IN := FALSE; END_IF
	timTimout_ReadAds(IN:= , PT:= T#30S, Q=> , ET=> );	

IF iState_WriteAds <> 0 AND iState_WriteAds <> -1 THEN timTimout_WriteAds.IN := TRUE; ELSE timTimout_WriteAds.IN := FALSE; END_IF
	timTimout_WriteAds(IN:= , PT:= T#30S, Q=> , ET=> );	
	
//Back to init if the search fb is busy
FPInitSendError(CLK:= Lynus_Standards.GVL_Communicator.arrInterfaceInfoValueSendTo[byReadWriteArrayNumber].bErrorSending, Q=> );
	IF FPInitSendError.Q THEN iState_ReadAds := -10; iState_WriteAds := -2; END_IF 

//Number for Loop of exists symbols
udiNumberLoopFull_ReadAds := Lynus_Standards.GVL_Communicator.arrCounterVariableInArray[byReadWriteArrayNumber];
	udiNumberLoopFull_ReadAds := LIMIT(1,udiNumberLoopFull_ReadAds,Lynus_Standards.Constants_Communicator.udiArraySizeMarkedSymobls);

udiNumberLoopHalf_ReadAds := STRING_TO_UDINT(LREAL_TO_FMTSTR((UDINT_TO_LREAL(udiNumberLoopFull_ReadAds) / 2),0,TRUE));
	udiNumberLoopHalf_ReadAds := LIMIT(1,udiNumberLoopHalf_ReadAds,STRING_TO_UDINT(LREAL_TO_FMTSTR((UDINT_TO_LREAL(udiNumberLoopFull_ReadAds) / 2),0,TRUE)));	
	
//Data write over ADS

CASE iState_WriteAds OF
	
	-2://Reset Write ADS (When deleting the array, conserve resources because the code must also work on small PLCs)
		Lynus_Standards.GVL_Communicator.arrInterfaceInfoValueWriteTo[byReadWriteArrayNumber].bWriteNewValue := FALSE; Lynus_Standards.GVL_Communicator.arrInterfaceInfoValueWriteTo[byReadWriteArrayNumber].bBusy := FALSE; Lynus_Standards.GVL_Communicator.arrInterfaceInfoValueWriteTo[byReadWriteArrayNumber].bErrorWrite := FALSE;
			bError_WriteAds := FALSE; bValueValid_WriteAds := FALSE;
				MEMCPY(ADR(arrBufferWrite_WriteAds),ADR(arrBufferWriteDefault_WriteAds),SIZEOF(arrBufferWrite_WriteAds));
					uiInternError_WriteAds := 0; byCounterEncodeString_WriteAds := 0; udiDate_WriteAds := 0; uiSizeToWrite_WriteAds := 0; byCounterReceivedValueOK_WriteAds := 0; uiCounterEncodeString_WriteAds := 0; uliDate_WriteAds := 0;
						byCounterWaitInStep_WriteAds := 0; dwVarHndl_WriteAds := 0;

		iState_WriteAds := -1;

	-1://Wait from info symbol function (When deleting the array, conserve resources because the code must also work on small PLCs)
		IF NOT Lynus_Standards.GVL_Communicator.bBusyInfoAlVariables AND NOT Lynus_Standards.GVL_Communicator.bErrorInfoAlVariables AND Lynus_Standards.GVL_Communicator.bInfoAlVariablesOK AND NOT Lynus_Standards.GVL_Communicator.arrInterfaceInfoValueSendTo[byReadWriteArrayNumber].bErrorSending AND
			bFirstReadCycleDone_ReadAds AND Lynus_Standards.GVL_Communicator.arrInterfaceInfoValueWriteTo[byReadWriteArrayNumber].bSendFunctionOK THEN 
				iState_WriteAds := 0;
		END_IF

	0://Init and clear write array befor wirte the new value (When deleting the array, conserve resources because the code must also work on small PLCs)
		Lynus_Standards.GVL_Communicator.arrInterfaceInfoValueWriteTo[byReadWriteArrayNumber].bErrorWrite := FALSE;
			arrCounterWriteValueInArray_WriteAds[1] := 0; arrCounterWriteValueInArray_WriteAds[2] := 0; arrCounterWriteValueInArray_WriteAds[3] := 0; arrCounterWriteValueInArray_WriteAds[4] := 0; arrCounterWriteValueInArray_WriteAds[5] := 0;
				arrCounterWriteValueInArray_WriteAds[6] := 0; arrCounterWriteValueInArray_WriteAds[7] := 0; arrCounterWriteValueInArray_WriteAds[8] := 0;
					rRealValueCheckBeforWrite_WriteAds := 0; lrRealValueCheckBeforWrite_WriteAds := 0; 
	
		IF Lynus_Standards.GVL_Communicator.arrInterfaceInfoValueWriteTo[byReadWriteArrayNumber].bWriteNewValue AND Lynus_Standards.GVL_Communicator.arrInterfaceInfoValueWriteTo[byReadWriteArrayNumber].sFullSymbolName <> '' THEN 
			iState_WriteAds := 1; 
				Lynus_Standards.GVL_Communicator.arrInterfaceInfoValueWriteTo[byReadWriteArrayNumber].bBusy := TRUE;
					MEMCPY(ADR(arrBufferWrite_WriteAds),ADR(arrBufferWriteDefault_WriteAds),SIZEOF(arrBufferWrite_WriteAds));
		END_IF

	1://Open var handle (When deleting the array, conserve resources because the code must also work on small PLCs)
		fbADSREADWRITE_WriteAds.WRITELEN := SIZEOF(Lynus_Standards.GVL_Communicator.arrInterfaceInfoValueWriteTo[byReadWriteArrayNumber].sFullSymbolName); 	
			fbADSREADWRITE_WriteAds.SRCADDR := ADR(Lynus_Standards.GVL_Communicator.arrInterfaceInfoValueWriteTo[byReadWriteArrayNumber].sFullSymbolName);
				fbADSREADWRITE_WriteAds.WRTRD := TRUE;	
		
		IF NOT fbADSREADWRITE_WriteAds.BUSY THEN byCounterWaitInStep_WriteAds := byCounterWaitInStep_WriteAds + 1; END_IF  		
	
		IF NOT fbADSREADWRITE_WriteAds.BUSY AND NOT fbADSREADWRITE_WriteAds.ERR AND byCounterWaitInStep_WriteAds >= byStaticValueWaitInStep AND dwVarHndl_WriteAds <> 0 THEN byCounterWaitInStep_WriteAds := 0; fbADSREADWRITE_WriteAds.WRTRD := FALSE; iState_WriteAds := 2; END_IF 
		
			IF FPErrorReadWrite_WriteAds.Q OR timTimout_WriteAds.Q THEN iState_WriteAds := 200; END_IF
			
